LIN {X 98.327,Y 109.227,Z 74.500,A 180.000,B 0.000,C 180.000} C_DIS
LIN {X 98.684,Y 109.197,Z 74.500,A 180.000,B 0.000,C 180.000} C_DIS
LIN {X 98.863,Y 109.180,Z 74.500,A 180.000,B 0.000,C 180.000} C_DIS
LIN {X 99.042,Y 109.155,Z 74.500,A 180.000,B 0.000,C 180.000} C_DIS
LIN {X 99.221,Y 109.129,Z 74.500,A 180.000,B 0.000,C 180.000} C_DIS
LIN {X 99.399,Y 109.104,Z 74.500,A 180.000,B 0.000,C 180.000} C_DIS
LIN {X 99.578,Y 109.071,Z 74.500,A 180.000,B 0.000,C 180.000} C_DIS
LIN {X 99.672,Y 109.053,Z 74.500,A 180.000,B 0.000,C 180.000} C_DIS
LIN {X 99.936,Y 109.000,Z 74.500,A 180.000,B 0.000,C 180.000} C_DIS
LIN {X 100.114,Y 108.964,Z 74.500,A 180.000,B 0.000,C 180.000} C_DIS
LIN {X 100.293,Y 108.920,Z 74.500,A 180.000,B 0.000,C 180.000} C_DIS
LIN {X 100.651,Y 108.828,Z 74.500,A 180.000,B 0.000,C 180.000} C_DIS
LIN {X 100.829,Y 108.776,Z 74.500,A 180.000,B 0.000,C 180.000} C_DIS
LIN {X 101.187,Y 108.662,Z 74.500,A 180.000,B 0.000,C 180.000} C_DIS
LIN {X 101.366,Y 108.604,Z 74.500,A 180.000,B 0.000,C 180.000} C_DIS
LIN {X 101.545,Y 108.539,Z 74.500,A 180.000,B 0.000,C 180.000} C_DIS
LIN {X 101.902,Y 108.403,Z 74.500,A 180.000,B 0.000,C 180.000} C_DIS
LIN {X 102.060,Y 108.338,Z 74.500,A 180.000,B 0.000,C 180.000} C_DIS
LIN {X 102.459,Y 108.159,Z 74.500,A 180.000,B 0.000,C 180.000} C_DIS
LIN {X 102.617,Y 108.086,Z 74.500,A 180.000,B 0.000,C 180.000} C_DIS
LIN {X 102.796,Y 107.996,Z 74.500,A 180.000,B 0.000,C 180.000} C_DIS
LIN {X 102.975,Y 107.903,Z 74.500,A 180.000,B 0.000,C 180.000} C_DIS
LIN {X 103.153,Y 107.811,Z 74.500,A 180.000,B 0.000,C 180.000} C_DIS
LIN {X 103.171,Y 107.802,Z 74.500,A 180.000,B 0.000,C 180.000} C_DIS
LIN {X 103.332,Y 107.708,Z 74.500,A 180.000,B 0.000,C 180.000} C_DIS
LIN {X 103.511,Y 107.602,Z 74.500,A 180.000,B 0.000,C 180.000} C_DIS
LIN {X 103.690,Y 107.497,Z 74.500,A 180.000,B 0.000,C 180.000} C_DIS
LIN {X 103.773,Y 107.444,Z 74.500,A 180.000,B 0.000,C 180.000} C_DIS
LIN {X 103.869,Y 107.382,Z 74.500,A 180.000,B 0.000,C 180.000} C_DIS
LIN {X 104.226,Y 107.144,Z 74.500,A 180.000,B 0.000,C 180.000} C_DIS
LIN {X 104.310,Y 107.086,Z 74.500,A 180.000,B 0.000,C 180.000} C_DIS
LIN {X 104.405,Y 107.016,Z 74.500,A 180.000,B 0.000,C 180.000} C_DIS
LIN {X 104.584,Y 106.882,Z 74.500,A 180.000,B 0.000,C 180.000} C_DIS
LIN {X 104.762,Y 106.747,Z 74.500,A 180.000,B 0.000,C 180.000} C_DIS
LIN {X 104.786,Y 106.729,Z 74.500,A 180.000,B 0.000,C 180.000} C_DIS
LIN {X 104.941,Y 106.601,Z 74.500,A 180.000,B 0.000,C 180.000} C_DIS
LIN {X 105.299,Y 106.300,Z 74.500,A 180.000,B 0.000,C 180.000} C_DIS
LIN {X 105.417,Y 106.193,Z 74.500,A 180.000,B 0.000,C 180.000} C_DIS
LIN {X 105.656,Y 105.967,Z 74.500,A 180.000,B 0.000,C 180.000} C_DIS
LIN {X 105.794,Y 105.835,Z 74.500,A 180.000,B 0.000,C 180.000} C_DIS
LIN {X 105.835,Y 105.793,Z 74.500,A 180.000,B 0.000,C 180.000} C_DIS
LIN {X 105.965,Y 105.656,Z 74.500,A 180.000,B 0.000,C 180.000} C_DIS
LIN {X 106.134,Y 105.477,Z 74.500,A 180.000,B 0.000,C 180.000} C_DIS
LIN {X 106.193,Y 105.415,Z 74.500,A 180.000,B 0.000,C 180.000} C_DIS
LIN {X 106.300,Y 105.299,Z 74.500,A 180.000,B 0.000,C 180.000} C_DIS
LIN {X 106.371,Y 105.215,Z 74.500,A 180.000,B 0.000,C 180.000} C_DIS
LIN {X 106.603,Y 104.941,Z 74.500,A 180.000,B 0.000,C 180.000} C_DIS
LIN {X 106.729,Y 104.786,Z 74.500,A 180.000,B 0.000,C 180.000} C_DIS
LIN {X 107.015,Y 104.405,Z 74.500,A 180.000,B 0.000,C 180.000} C_DIS
LIN {X 107.086,Y 104.308,Z 74.500,A 180.000,B 0.000,C 180.000} C_DIS
LIN {X 107.144,Y 104.226,Z 74.500,A 180.000,B 0.000,C 180.000} C_DIS
LIN {X 107.265,Y 104.045,Z 74.500,A 180.000,B 0.000,C 180.000} C_DIS
LIN {X 107.383,Y 103.869,Z 74.500,A 180.000,B 0.000,C 180.000} C_DIS
LIN {X 107.444,Y 103.776,Z 74.500,A 180.000,B 0.000,C 180.000} C_DIS
LIN {X 107.497,Y 103.690,Z 74.500,A 180.000,B 0.000,C 180.000} C_DIS
LIN {X 107.708,Y 103.332,Z 74.500,A 180.000,B 0.000,C 180.000} C_DIS
LIN {X 107.802,Y 103.167,Z 74.500,A 180.000,B 0.000,C 180.000} C_DIS
LIN {X 107.809,Y 103.153,Z 74.500,A 180.000,B 0.000,C 180.000} C_DIS
LIN {X 107.903,Y 102.975,Z 74.500,A 180.000,B 0.000,C 180.000} C_DIS
LIN {X 107.995,Y 102.796,Z 74.500,A 180.000,B 0.000,C 180.000} C_DIS
LIN {X 108.087,Y 102.617,Z 74.500,A 180.000,B 0.000,C 180.000} C_DIS
LIN {X 108.159,Y 102.461,Z 74.500,A 180.000,B 0.000,C 180.000} C_DIS
LIN {X 108.249,Y 102.260,Z 74.500,A 180.000,B 0.000,C 180.000} C_DIS
LIN {X 108.329,Y 102.081,Z 74.500,A 180.000,B 0.000,C 180.000} C_DIS
LIN {X 108.338,Y 102.061,Z 74.500,A 180.000,B 0.000,C 180.000} C_DIS
LIN {X 108.402,Y 101.902,Z 74.500,A 180.000,B 0.000,C 180.000} C_DIS
LIN {X 108.470,Y 101.723,Z 74.500,A 180.000,B 0.000,C 180.000} C_DIS
LIN {X 108.538,Y 101.545,Z 74.500,A 180.000,B 0.000,C 180.000} C_DIS
LIN {X 108.605,Y 101.366,Z 74.500,A 180.000,B 0.000,C 180.000} C_DIS
LIN {X 108.663,Y 101.187,Z 74.500,A 180.000,B 0.000,C 180.000} C_DIS
LIN {X 108.720,Y 101.008,Z 74.500,A 180.000,B 0.000,C 180.000} C_DIS
LIN {X 108.777,Y 100.829,Z 74.500,A 180.000,B 0.000,C 180.000} C_DIS
LIN {X 108.826,Y 100.651,Z 74.500,A 180.000,B 0.000,C 180.000} C_DIS
LIN {X 108.919,Y 100.293,Z 74.500,A 180.000,B 0.000,C 180.000} C_DIS
LIN {X 108.964,Y 100.114,Z 74.500,A 180.000,B 0.000,C 180.000} C_DIS
LIN {X 109.002,Y 99.936,Z 74.500,A 180.000,B 0.000,C 180.000} C_DIS
LIN {X 109.073,Y 99.578,Z 74.500,A 180.000,B 0.000,C 180.000} C_DIS
LIN {X 109.103,Y 99.399,Z 74.500,A 180.000,B 0.000,C 180.000} C_DIS
LIN {X 109.154,Y 99.042,Z 74.500,A 180.000,B 0.000,C 180.000} C_DIS
LIN {X 109.178,Y 98.863,Z 74.500,A 180.000,B 0.000,C 180.000} C_DIS
LIN {X 109.197,Y 98.684,Z 74.500,A 180.000,B 0.000,C 180.000} C_DIS
LIN {X 109.232,Y 98.279,Z 74.500,A 180.000,B 0.000,C 180.000} C_DIS
LIN {X 109.241,Y 98.148,Z 74.500,A 180.000,B 0.000,C 180.000} C_DIS
LIN {X 109.247,Y 97.969,Z 74.500,A 180.000,B 0.000,C 180.000} C_DIS
LIN {X 109.252,Y 97.790,Z 74.500,A 180.000,B 0.000,C 180.000} C_DIS
LIN {X 109.257,Y 97.612,Z 74.500,A 180.000,B 0.000,C 180.000} C_DIS
LIN {X 109.257,Y 97.433,Z 74.500,A 180.000,B 0.000,C 180.000} C_DIS
LIN {X 109.253,Y 97.254,Z 74.500,A 180.000,B 0.000,C 180.000} C_DIS
LIN {X 109.248,Y 97.075,Z 74.500,A 180.000,B 0.000,C 180.000} C_DIS
LIN {X 109.243,Y 96.897,Z 74.500,A 180.000,B 0.000,C 180.000} C_DIS
LIN {X 109.232,Y 96.721,Z 74.500,A 180.000,B 0.000,C 180.000} C_DIS
LIN {X 109.201,Y 96.360,Z 74.500,A 180.000,B 0.000,C 180.000} C_DIS
LIN {X 109.184,Y 96.181,Z 74.500,A 180.000,B 0.000,C 180.000} C_DIS
LIN {X 109.160,Y 96.003,Z 74.500,A 180.000,B 0.000,C 180.000} C_DIS
LIN {X 109.110,Y 95.645,Z 74.500,A 180.000,B 0.000,C 180.000} C_DIS
LIN {X 109.081,Y 95.466,Z 74.500,A 180.000,B 0.000,C 180.000} C_DIS
LIN {X 109.053,Y 95.322,Z 74.500,A 180.000,B 0.000,C 180.000} C_DIS
LIN {X 109.010,Y 95.109,Z 74.500,A 180.000,B 0.000,C 180.000} C_DIS
LIN {X 108.974,Y 94.930,Z 74.500,A 180.000,B 0.000,C 180.000} C_DIS
LIN {X 108.930,Y 94.751,Z 74.500,A 180.000,B 0.000,C 180.000} C_DIS
LIN {X 108.838,Y 94.394,Z 74.500,A 180.000,B 0.000,C 180.000} C_DIS
LIN {X 108.791,Y 94.215,Z 74.500,A 180.000,B 0.000,C 180.000} C_DIS
LIN {X 108.734,Y 94.036,Z 74.500,A 180.000,B 0.000,C 180.000} C_DIS
LIN {X 108.677,Y 93.857,Z 74.500,A 180.000,B 0.000,C 180.000} C_DIS
LIN {X 108.620,Y 93.679,Z 74.500,A 180.000,B 0.000,C 180.000} C_DIS
LIN {X 108.555,Y 93.500,Z 74.500,A 180.000,B 0.000,C 180.000} C_DIS
LIN {X 108.419,Y 93.142,Z 74.500,A 180.000,B 0.000,C 180.000} C_DIS
LIN {X 108.348,Y 92.964,Z 74.500,A 180.000,B 0.000,C 180.000} C_DIS
LIN {X 108.338,Y 92.939,Z 74.500,A 180.000,B 0.000,C 180.000} C_DIS
LIN {X 108.269,Y 92.785,Z 74.500,A 180.000,B 0.000,C 180.000} C_DIS
LIN {X 108.159,Y 92.539,Z 74.500,A 180.000,B 0.000,C 180.000} C_DIS
LIN {X 108.109,Y 92.427,Z 74.500,A 180.000,B 0.000,C 180.000} C_DIS
LIN {X 108.018,Y 92.249,Z 74.500,A 180.000,B 0.000,C 180.000} C_DIS
LIN {X 107.926,Y 92.070,Z 74.500,A 180.000,B 0.000,C 180.000} C_DIS
LIN {X 107.833,Y 91.891,Z 74.500,A 180.000,B 0.000,C 180.000} C_DIS
LIN {X 107.802,Y 91.833,Z 74.500,A 180.000,B 0.000,C 180.000} C_DIS
LIN {X 107.734,Y 91.712,Z 74.500,A 180.000,B 0.000,C 180.000} C_DIS
LIN {X 107.523,Y 91.355,Z 74.500,A 180.000,B 0.000,C 180.000} C_DIS
LIN {X 107.444,Y 91.224,Z 74.500,A 180.000,B 0.000,C 180.000} C_DIS
LIN {X 107.413,Y 91.176,Z 74.500,A 180.000,B 0.000,C 180.000} C_DIS
LIN {X 107.174,Y 90.818,Z 74.500,A 180.000,B 0.000,C 180.000} C_DIS
LIN {X 107.086,Y 90.692,Z 74.500,A 180.000,B 0.000,C 180.000} C_DIS
LIN {X 107.048,Y 90.640,Z 74.500,A 180.000,B 0.000,C 180.000} C_DIS
LIN {X 106.914,Y 90.461,Z 74.500,A 180.000,B 0.000,C 180.000} C_DIS
LIN {X 106.729,Y 90.214,Z 74.500,A 180.000,B 0.000,C 180.000} C_DIS
LIN {X 106.640,Y 90.103,Z 74.500,A 180.000,B 0.000,C 180.000} C_DIS
LIN {X 106.338,Y 89.746,Z 74.500,A 180.000,B 0.000,C 180.000} C_DIS
LIN {X 106.193,Y 89.585,Z 74.500,A 180.000,B 0.000,C 180.000} C_DIS
LIN {X 106.176,Y 89.567,Z 74.500,A 180.000,B 0.000,C 180.000} C_DIS
LIN {X 106.007,Y 89.388,Z 74.500,A 180.000,B 0.000,C 180.000} C_DIS
LIN {X 105.838,Y 89.209,Z 74.500,A 180.000,B 0.000,C 180.000} C_DIS
LIN {X 105.835,Y 89.207,Z 74.500,A 180.000,B 0.000,C 180.000} C_DIS
LIN {X 105.656,Y 89.033,Z 74.500,A 180.000,B 0.000,C 180.000} C_DIS
LIN {X 105.464,Y 88.852,Z 74.500,A 180.000,B 0.000,C 180.000} C_DIS
LIN {X 105.299,Y 88.700,Z 74.500,A 180.000,B 0.000,C 180.000} C_DIS
LIN {X 104.941,Y 88.399,Z 74.500,A 180.000,B 0.000,C 180.000} C_DIS
LIN {X 104.841,Y 88.316,Z 74.500,A 180.000,B 0.000,C 180.000} C_DIS
LIN {X 104.762,Y 88.253,Z 74.500,A 180.000,B 0.000,C 180.000} C_DIS
LIN {X 104.608,Y 88.137,Z 74.500,A 180.000,B 0.000,C 180.000} C_DIS
LIN {X 104.371,Y 87.958,Z 74.500,A 180.000,B 0.000,C 180.000} C_DIS
LIN {X 104.226,Y 87.856,Z 74.500,A 180.000,B 0.000,C 180.000} C_DIS
LIN {X 103.869,Y 87.618,Z 74.500,A 180.000,B 0.000,C 180.000} C_DIS
LIN {X 103.843,Y 87.601,Z 74.500,A 180.000,B 0.000,C 180.000} C_DIS
LIN {X 103.690,Y 87.503,Z 74.500,A 180.000,B 0.000,C 180.000} C_DIS
LIN {X 103.552,Y 87.422,Z 74.500,A 180.000,B 0.000,C 180.000} C_DIS
LIN {X 103.249,Y 87.243,Z 74.500,A 180.000,B 0.000,C 180.000} C_DIS
LIN {X 103.153,Y 87.189,Z 74.500,A 180.000,B 0.000,C 180.000} C_DIS
LIN {X 102.975,Y 87.097,Z 74.500,A 180.000,B 0.000,C 180.000} C_DIS
LIN {X 102.796,Y 87.004,Z 74.500,A 180.000,B 0.000,C 180.000} C_DIS
LIN {X 102.617,Y 86.914,Z 74.500,A 180.000,B 0.000,C 180.000} C_DIS
LIN {X 102.556,Y 86.885,Z 74.500,A 180.000,B 0.000,C 180.000} C_DIS
LIN {X 102.438,Y 86.832,Z 74.500,A 180.000,B 0.000,C 180.000} C_DIS
LIN {X 102.191,Y 86.721,Z 74.500,A 180.000,B 0.000,C 180.000} C_DIS
; Link Move Starts
LIN {X 101.924,Y 86.603,Z 74.500,A 180.000,B 0.000,C 180.000} C_DIS
LIN {X 101.633,Y 86.492,Z 74.499,A 180.000,B 0.000,C 180.000} C_DIS
LIN {X 101.360,Y 86.390,Z 74.498,A 180.000,B 0.000,C 180.000} C_DIS
LIN {X 101.062,Y 86.294,Z 74.496,A 180.000,B 0.000,C 180.000} C_DIS
LIN {X 100.768,Y 86.200,Z 74.494,A 180.000,B 0.000,C 180.000} C_DIS
LIN {X 100.483,Y 86.123,Z 74.492,A 180.000,B 0.000,C 180.000} C_DIS
LIN {X 100.187,Y 86.045,Z 74.489,A 180.000,B 0.000,C 180.000} C_DIS
LIN {X 99.896,Y 85.983,Z 74.486,A 180.000,B 0.000,C 180.000} C_DIS
LIN {X 99.589,Y 85.920,Z 74.482,A 180.000,B 0.000,C 180.000} C_DIS
LIN {X 99.302,Y 85.870,Z 74.478,A 180.000,B 0.000,C 180.000} C_DIS
LIN {X 98.991,Y 85.824,Z 74.474,A 180.000,B 0.000,C 180.000} C_DIS
LIN {X 98.702,Y 85.788,Z 74.469,A 180.000,B 0.000,C 180.000} C_DIS
LIN {X 98.546,Y 85.773,Z 74.467,A 180.000,B 0.000,C 180.000} C_DIS
LIN {X 98.390,Y 85.759,Z 74.464,A 180.000,B 0.000,C 180.000} C_DIS
LIN {X 98.244,Y 85.746,Z 74.461,A 180.000,B 0.000,C 180.000} C_DIS
LIN {X 98.098,Y 85.736,Z 74.459,A 180.000,B 0.000,C 180.000} C_DIS
LIN {X 97.942,Y 85.729,Z 74.456,A 180.000,B 0.000,C 180.000} C_DIS
LIN {X 97.786,Y 85.724,Z 74.453,A 180.000,B 0.000,C 180.000} C_DIS
LIN {X 97.633,Y 85.718,Z 74.450,A 180.000,B 0.000,C 180.000} C_DIS
LIN {X 97.480,Y 85.714,Z 74.447,A 180.000,B 0.000,C 180.000} C_DIS
LIN {X 97.331,Y 85.716,Z 74.443,A 180.000,B 0.000,C 180.000} C_DIS
LIN {X 97.181,Y 85.719,Z 74.440,A 180.000,B 0.000,C 180.000} C_DIS
LIN {X 97.030,Y 85.721,Z 74.437,A 180.000,B 0.000,C 180.000} C_DIS
LIN {X 96.880,Y 85.725,Z 74.433,A 180.000,B 0.000,C 180.000} C_DIS
LIN {X 96.728,Y 85.733,Z 74.430,A 180.000,B 0.000,C 180.000} C_DIS
LIN {X 96.576,Y 85.744,Z 74.426,A 180.000,B 0.000,C 180.000} C_DIS
LIN {X 96.419,Y 85.756,Z 74.422,A 180.000,B 0.000,C 180.000} C_DIS
LIN {X 96.262,Y 85.767,Z 74.418,A 180.000,B 0.000,C 180.000} C_DIS
LIN {X 96.117,Y 85.781,Z 74.415,A 180.000,B 0.000,C 180.000} C_DIS
LIN {X 95.973,Y 85.799,Z 74.411,A 180.000,B 0.000,C 180.000} C_DIS
LIN {X 95.818,Y 85.819,Z 74.407,A 180.000,B 0.000,C 180.000} C_DIS
LIN {X 95.663,Y 85.839,Z 74.403,A 180.000,B 0.000,C 180.000} C_DIS
LIN {X 95.517,Y 85.860,Z 74.399,A 180.000,B 0.000,C 180.000} C_DIS
LIN {X 95.370,Y 85.886,Z 74.394,A 180.000,B 0.000,C 180.000} C_DIS
LIN {X 95.217,Y 85.915,Z 74.390,A 180.000,B 0.000,C 180.000} C_DIS
LIN {X 95.063,Y 85.943,Z 74.386,A 180.000,B 0.000,C 180.000} C_DIS
LIN {X 94.918,Y 85.970,Z 74.381,A 180.000,B 0.000,C 180.000} C_DIS
LIN {X 94.775,Y 86.001,Z 74.377,A 180.000,B 0.000,C 180.000} C_DIS
LIN {X 94.622,Y 86.038,Z 74.372,A 180.000,B 0.000,C 180.000} C_DIS
LIN {X 94.470,Y 86.075,Z 74.368,A 180.000,B 0.000,C 180.000} C_DIS
LIN {X 94.323,Y 86.110,Z 74.363,A 180.000,B 0.000,C 180.000} C_DIS
LIN {X 94.177,Y 86.150,Z 74.358,A 180.000,B 0.000,C 180.000} C_DIS
LIN {X 94.031,Y 86.194,Z 74.353,A 180.000,B 0.000,C 180.000} C_DIS
LIN {X 93.885,Y 86.238,Z 74.348,A 180.000,B 0.000,C 180.000} C_DIS
LIN {X 93.740,Y 86.282,Z 74.343,A 180.000,B 0.000,C 180.000} C_DIS
LIN {X 93.594,Y 86.327,Z 74.339,A 180.000,B 0.000,C 180.000} C_DIS
LIN {X 93.522,Y 86.351,Z 74.336,A 180.000,B 0.000,C 180.000} C_DIS
LIN {X 93.451,Y 86.377,Z 74.333,A 180.000,B 0.000,C 180.000} C_DIS
LIN {X 93.379,Y 86.403,Z 74.331,A 180.000,B 0.000,C 180.000} C_DIS
LIN {X 93.236,Y 86.455,Z 74.326,A 180.000,B 0.000,C 180.000} C_DIS
LIN {X 93.164,Y 86.481,Z 74.323,A 180.000,B 0.000,C 180.000} C_DIS
LIN {X 93.092,Y 86.508,Z 74.321,A 180.000,B 0.000,C 180.000} C_DIS
LIN {X 93.020,Y 86.534,Z 74.318,A 180.000,B 0.000,C 180.000} C_DIS
LIN {X 92.950,Y 86.561,Z 74.315,A 180.000,B 0.000,C 180.000} C_DIS
LIN {X 92.880,Y 86.591,Z 74.313,A 180.000,B 0.000,C 180.000} C_DIS
LIN {X 92.525,Y 86.743,Z 74.299,A 180.000,B 0.000,C 180.000} C_DIS
LIN {X 92.453,Y 86.774,Z 74.296,A 180.000,B 0.000,C 180.000} C_DIS
LIN {X 92.385,Y 86.804,Z 74.294,A 180.000,B 0.000,C 180.000} C_DIS
LIN {X 92.318,Y 86.835,Z 74.291,A 180.000,B 0.000,C 180.000} C_DIS
LIN {X 92.251,Y 86.867,Z 74.289,A 180.000,B 0.000,C 180.000} C_DIS
LIN {X 92.185,Y 86.899,Z 74.286,A 180.000,B 0.000,C 180.000} C_DIS
LIN {X 92.044,Y 86.969,Z 74.281,A 180.000,B 0.000,C 180.000} C_DIS
LIN {X 91.837,Y 87.072,Z 74.273,A 180.000,B 0.000,C 180.000} C_DIS
LIN {X 91.771,Y 87.106,Z 74.270,A 180.000,B 0.000,C 180.000} C_DIS
LIN {X 91.706,Y 87.141,Z 74.267,A 180.000,B 0.000,C 180.000} C_DIS
LIN {X 91.642,Y 87.177,Z 74.265,A 180.000,B 0.000,C 180.000} C_DIS
LIN {X 91.505,Y 87.255,Z 74.259,A 180.000,B 0.000,C 180.000} C_DIS
LIN {X 91.303,Y 87.370,Z 74.251,A 180.000,B 0.000,C 180.000} C_DIS
LIN {X 91.238,Y 87.407,Z 74.249,A 180.000,B 0.000,C 180.000} C_DIS
LIN {X 91.174,Y 87.446,Z 74.246,A 180.000,B 0.000,C 180.000} C_DIS
LIN {X 91.110,Y 87.485,Z 74.243,A 180.000,B 0.000,C 180.000} C_DIS
LIN {X 91.045,Y 87.527,Z 74.241,A 180.000,B 0.000,C 180.000} C_DIS
LIN {X 90.914,Y 87.611,Z 74.235,A 180.000,B 0.000,C 180.000} C_DIS
LIN {X 90.849,Y 87.654,Z 74.233,A 180.000,B 0.000,C 180.000} C_DIS
LIN {X 90.722,Y 87.735,Z 74.227,A 180.000,B 0.000,C 180.000} C_DIS
LIN {X 90.658,Y 87.776,Z 74.225,A 180.000,B 0.000,C 180.000} C_DIS
LIN {X 90.596,Y 87.819,Z 74.222,A 180.000,B 0.000,C 180.000} C_DIS
LIN {X 90.533,Y 87.864,Z 74.219,A 180.000,B 0.000,C 180.000} C_DIS
LIN {X 90.408,Y 87.955,Z 74.214,A 180.000,B 0.000,C 180.000} C_DIS
LIN {X 90.346,Y 88.000,Z 74.211,A 180.000,B 0.000,C 180.000} C_DIS
LIN {X 90.223,Y 88.090,Z 74.206,A 180.000,B 0.000,C 180.000} C_DIS
LIN {X 90.161,Y 88.134,Z 74.203,A 180.000,B 0.000,C 180.000} C_DIS
LIN {X 90.100,Y 88.180,Z 74.201,A 180.000,B 0.000,C 180.000} C_DIS
LIN {X 90.040,Y 88.228,Z 74.198,A 180.000,B 0.000,C 180.000} C_DIS
LIN {X 89.980,Y 88.276,Z 74.195,A 180.000,B 0.000,C 180.000} C_DIS
LIN {X 89.800,Y 88.423,Z 74.187,A 180.000,B 0.000,C 180.000} C_DIS
LIN {X 89.678,Y 88.523,Z 74.182,A 180.000,B 0.000,C 180.000} C_DIS
LIN {X 89.617,Y 88.573,Z 74.179,A 180.000,B 0.000,C 180.000} C_DIS
LIN {X 89.560,Y 88.620,Z 74.176,A 180.000,B 0.000,C 180.000} C_DIS
LIN {X 89.504,Y 88.669,Z 74.174,A 180.000,B 0.000,C 180.000} C_DIS
LIN {X 89.449,Y 88.719,Z 74.171,A 180.000,B 0.000,C 180.000} C_DIS
LIN {X 89.394,Y 88.770,Z 74.168,A 180.000,B 0.000,C 180.000} C_DIS
LIN {X 89.279,Y 88.875,Z 74.163,A 180.000,B 0.000,C 180.000} C_DIS
LIN {X 89.163,Y 88.981,Z 74.157,A 180.000,B 0.000,C 180.000} C_DIS
LIN {X 89.108,Y 89.032,Z 74.155,A 180.000,B 0.000,C 180.000} C_DIS
LIN {X 89.054,Y 89.084,Z 74.152,A 180.000,B 0.000,C 180.000} C_DIS
LIN {X 89.002,Y 89.138,Z 74.150,A 180.000,B 0.000,C 180.000} C_DIS
LIN {X 88.894,Y 89.248,Z 74.144,A 180.000,B 0.000,C 180.000} C_DIS
LIN {X 88.730,Y 89.417,Z 74.136,A 180.000,B 0.000,C 180.000} C_DIS
LIN {X 88.677,Y 89.470,Z 74.133,A 180.000,B 0.000,C 180.000} C_DIS
LIN {X 88.625,Y 89.524,Z 74.131,A 180.000,B 0.000,C 180.000} C_DIS
LIN {X 88.574,Y 89.578,Z 74.128,A 180.000,B 0.000,C 180.000} C_DIS
LIN {X 88.525,Y 89.634,Z 74.126,A 180.000,B 0.000,C 180.000} C_DIS
LIN {X 88.369,Y 89.812,Z 74.117,A 180.000,B 0.000,C 180.000} C_DIS
LIN {X 88.268,Y 89.927,Z 74.112,A 180.000,B 0.000,C 180.000} C_DIS
LIN {X 88.219,Y 89.984,Z 74.109,A 180.000,B 0.000,C 180.000} C_DIS
LIN {X 88.171,Y 90.041,Z 74.107,A 180.000,B 0.000,C 180.000} C_DIS
LIN {X 88.124,Y 90.099,Z 74.104,A 180.000,B 0.000,C 180.000} C_DIS
LIN {X 87.979,Y 90.286,Z 74.096,A 180.000,B 0.000,C 180.000} C_DIS
LIN {X 87.835,Y 90.470,Z 74.088,A 180.000,B 0.000,C 180.000} C_DIS
LIN {X 87.788,Y 90.532,Z 74.085,A 180.000,B 0.000,C 180.000} C_DIS
LIN {X 87.741,Y 90.594,Z 74.082,A 180.000,B 0.000,C 180.000} C_DIS
LIN {X 87.697,Y 90.656,Z 74.080,A 180.000,B 0.000,C 180.000} C_DIS
LIN {X 87.653,Y 90.718,Z 74.077,A 180.000,B 0.000,C 180.000} C_DIS
LIN {X 87.433,Y 91.037,Z 74.063,A 180.000,B 0.000,C 180.000} C_DIS
LIN {X 87.389,Y 91.101,Z 74.061,A 180.000,B 0.000,C 180.000} C_DIS
LIN {X 87.347,Y 91.164,Z 74.058,A 180.000,B 0.000,C 180.000} C_DIS
LIN {X 87.308,Y 91.229,Z 74.055,A 180.000,B 0.000,C 180.000} C_DIS
LIN {X 87.106,Y 91.558,Z 74.042,A 180.000,B 0.000,C 180.000} C_DIS
LIN {X 87.065,Y 91.625,Z 74.039,A 180.000,B 0.000,C 180.000} C_DIS
LIN {X 87.027,Y 91.691,Z 74.037,A 180.000,B 0.000,C 180.000} C_DIS
LIN {X 86.990,Y 91.756,Z 74.034,A 180.000,B 0.000,C 180.000} C_DIS
LIN {X 86.953,Y 91.822,Z 74.031,A 180.000,B 0.000,C 180.000} C_DIS
LIN {X 86.733,Y 92.233,Z 74.015,A 180.000,B 0.000,C 180.000} C_DIS
LIN {X 86.698,Y 92.300,Z 74.012,A 180.000,B 0.000,C 180.000} C_DIS
LIN {X 86.665,Y 92.368,Z 74.010,A 180.000,B 0.000,C 180.000} C_DIS
LIN {X 86.468,Y 92.789,Z 73.993,A 180.000,B 0.000,C 180.000} C_DIS
LIN {X 86.436,Y 92.858,Z 73.991,A 180.000,B 0.000,C 180.000} C_DIS
LIN {X 86.406,Y 92.928,Z 73.988,A 180.000,B 0.000,C 180.000} C_DIS
LIN {X 86.377,Y 92.999,Z 73.986,A 180.000,B 0.000,C 180.000} C_DIS
LIN {X 86.348,Y 93.071,Z 73.983,A 180.000,B 0.000,C 180.000} C_DIS
LIN {X 86.204,Y 93.432,Z 73.969,A 180.000,B 0.000,C 180.000} C_DIS
LIN {X 86.175,Y 93.502,Z 73.967,A 180.000,B 0.000,C 180.000} C_DIS
LIN {X 86.149,Y 93.574,Z 73.964,A 180.000,B 0.000,C 180.000} C_DIS
LIN {X 86.123,Y 93.648,Z 73.961,A 180.000,B 0.000,C 180.000} C_DIS
LIN {X 85.975,Y 94.089,Z 73.945,A 180.000,B 0.000,C 180.000} C_DIS
LIN {X 85.952,Y 94.162,Z 73.942,A 180.000,B 0.000,C 180.000} C_DIS
LIN {X 85.930,Y 94.237,Z 73.940,A 180.000,B 0.000,C 180.000} C_DIS
LIN {X 85.806,Y 94.690,Z 73.923,A 180.000,B 0.000,C 180.000} C_DIS
LIN {X 85.785,Y 94.766,Z 73.920,A 180.000,B 0.000,C 180.000} C_DIS
LIN {X 85.765,Y 94.839,Z 73.918,A 180.000,B 0.000,C 180.000} C_DIS
LIN {X 85.748,Y 94.913,Z 73.915,A 180.000,B 0.000,C 180.000} C_DIS
LIN {X 85.650,Y 95.370,Z 73.899,A 180.000,B 0.000,C 180.000} C_DIS
LIN {X 85.634,Y 95.444,Z 73.896,A 180.000,B 0.000,C 180.000} C_DIS
LIN {X 85.620,Y 95.519,Z 73.893,A 180.000,B 0.000,C 180.000} C_DIS
LIN {X 85.608,Y 95.595,Z 73.891,A 180.000,B 0.000,C 180.000} C_DIS
LIN {X 85.584,Y 95.748,Z 73.885,A 180.000,B 0.000,C 180.000} C_DIS
LIN {X 85.547,Y 95.981,Z 73.877,A 180.000,B 0.000,C 180.000} C_DIS
LIN {X 85.536,Y 96.057,Z 73.874,A 180.000,B 0.000,C 180.000} C_DIS
LIN {X 85.525,Y 96.132,Z 73.872,A 180.000,B 0.000,C 180.000} C_DIS
LIN {X 85.515,Y 96.208,Z 73.869,A 180.000,B 0.000,C 180.000} C_DIS
LIN {X 85.507,Y 96.284,Z 73.866,A 180.000,B 0.000,C 180.000} C_DIS
LIN {X 85.483,Y 96.519,Z 73.858,A 180.000,B 0.000,C 180.000} C_DIS
LIN {X 85.467,Y 96.674,Z 73.853,A 180.000,B 0.000,C 180.000} C_DIS
LIN {X 85.460,Y 96.750,Z 73.850,A 180.000,B 0.000,C 180.000} C_DIS
LIN {X 85.453,Y 96.827,Z 73.847,A 180.000,B 0.000,C 180.000} C_DIS
LIN {X 85.449,Y 96.904,Z 73.845,A 180.000,B 0.000,C 180.000} C_DIS
LIN {X 85.442,Y 97.060,Z 73.839,A 180.000,B 0.000,C 180.000} C_DIS
LIN {X 85.428,Y 97.371,Z 73.828,A 180.000,B 0.000,C 180.000} C_DIS
LIN {X 85.426,Y 97.449,Z 73.826,A 180.000,B 0.000,C 180.000} C_DIS
LIN {X 85.424,Y 97.526,Z 73.823,A 180.000,B 0.000,C 180.000} C_DIS
LIN {X 85.424,Y 97.604,Z 73.820,A 180.000,B 0.000,C 180.000} C_DIS
LIN {X 85.425,Y 97.682,Z 73.818,A 180.000,B 0.000,C 180.000} C_DIS
LIN {X 85.429,Y 98.070,Z 73.804,A 180.000,B 0.000,C 180.000} C_DIS
LIN {X 85.430,Y 98.147,Z 73.801,A 180.000,B 0.000,C 180.000} C_DIS
LIN {X 85.434,Y 98.225,Z 73.799,A 180.000,B 0.000,C 180.000} C_DIS
LIN {X 85.439,Y 98.304,Z 73.796,A 180.000,B 0.000,C 180.000} C_DIS
LIN {X 85.455,Y 98.538,Z 73.788,A 180.000,B 0.000,C 180.000} C_DIS
LIN {X 85.465,Y 98.694,Z 73.782,A 180.000,B 0.000,C 180.000} C_DIS
LIN {X 85.471,Y 98.773,Z 73.779,A 180.000,B 0.000,C 180.000} C_DIS
LIN {X 85.478,Y 98.849,Z 73.777,A 180.000,B 0.000,C 180.000} C_DIS
LIN {X 85.486,Y 98.926,Z 73.774,A 180.000,B 0.000,C 180.000} C_DIS
LIN {X 85.495,Y 99.003,Z 73.771,A 180.000,B 0.000,C 180.000} C_DIS
LIN {X 85.505,Y 99.080,Z 73.769,A 180.000,B 0.000,C 180.000} C_DIS
LIN {X 85.524,Y 99.236,Z 73.763,A 180.000,B 0.000,C 180.000} C_DIS
LIN {X 85.553,Y 99.468,Z 73.755,A 180.000,B 0.000,C 180.000} C_DIS
LIN {X 85.564,Y 99.545,Z 73.752,A 180.000,B 0.000,C 180.000} C_DIS
LIN {X 85.577,Y 99.621,Z 73.750,A 180.000,B 0.000,C 180.000} C_DIS
LIN {X 85.591,Y 99.697,Z 73.747,A 180.000,B 0.000,C 180.000} C_DIS
LIN {X 85.619,Y 99.852,Z 73.741,A 180.000,B 0.000,C 180.000} C_DIS
LIN {X 85.661,Y 100.083,Z 73.733,A 180.000,B 0.000,C 180.000} C_DIS
LIN {X 85.675,Y 100.159,Z 73.730,A 180.000,B 0.000,C 180.000} C_DIS
LIN {X 85.692,Y 100.235,Z 73.728,A 180.000,B 0.000,C 180.000} C_DIS
LIN {X 85.710,Y 100.310,Z 73.725,A 180.000,B 0.000,C 180.000} C_DIS
LIN {X 85.729,Y 100.386,Z 73.722,A 180.000,B 0.000,C 180.000} C_DIS
LIN {X 85.765,Y 100.539,Z 73.717,A 180.000,B 0.000,C 180.000} C_DIS
LIN {X 85.784,Y 100.616,Z 73.714,A 180.000,B 0.000,C 180.000} C_DIS
LIN {X 85.820,Y 100.768,Z 73.709,A 180.000,B 0.000,C 180.000} C_DIS
LIN {X 85.839,Y 100.843,Z 73.706,A 180.000,B 0.000,C 180.000} C_DIS
LIN {X 85.859,Y 100.919,Z 73.703,A 180.000,B 0.000,C 180.000} C_DIS
LIN {X 85.881,Y 100.994,Z 73.700,A 180.000,B 0.000,C 180.000} C_DIS
LIN {X 85.927,Y 101.143,Z 73.695,A 180.000,B 0.000,C 180.000} C_DIS
LIN {X 85.994,Y 101.368,Z 73.687,A 180.000,B 0.000,C 180.000} C_DIS
LIN {X 86.017,Y 101.443,Z 73.684,A 180.000,B 0.000,C 180.000} C_DIS
LIN {X 86.041,Y 101.517,Z 73.681,A 180.000,B 0.000,C 180.000} C_DIS
LIN {X 86.067,Y 101.591,Z 73.679,A 180.000,B 0.000,C 180.000} C_DIS
LIN {X 86.094,Y 101.664,Z 73.676,A 180.000,B 0.000,C 180.000} C_DIS
LIN {X 86.121,Y 101.738,Z 73.674,A 180.000,B 0.000,C 180.000} C_DIS
LIN {X 86.147,Y 101.811,Z 73.671,A 180.000,B 0.000,C 180.000} C_DIS
LIN {X 86.174,Y 101.885,Z 73.668,A 180.000,B 0.000,C 180.000} C_DIS
LIN {X 86.201,Y 101.958,Z 73.666,A 180.000,B 0.000,C 180.000} C_DIS
LIN {X 86.228,Y 102.032,Z 73.663,A 180.000,B 0.000,C 180.000} C_DIS
LIN {X 86.255,Y 102.105,Z 73.661,A 180.000,B 0.000,C 180.000} C_DIS
LIN {X 86.283,Y 102.178,Z 73.658,A 180.000,B 0.000,C 180.000} C_DIS
LIN {X 86.313,Y 102.250,Z 73.655,A 180.000,B 0.000,C 180.000} C_DIS
LIN {X 86.344,Y 102.322,Z 73.653,A 180.000,B 0.000,C 180.000} C_DIS
LIN {X 86.375,Y 102.394,Z 73.650,A 180.000,B 0.000,C 180.000} C_DIS
LIN {X 86.437,Y 102.539,Z 73.645,A 180.000,B 0.000,C 180.000} C_DIS
LIN {X 86.499,Y 102.683,Z 73.641,A 180.000,B 0.000,C 180.000} C_DIS
LIN {X 86.564,Y 102.825,Z 73.636,A 180.000,B 0.000,C 180.000} C_DIS
LIN {X 86.633,Y 102.965,Z 73.631,A 180.000,B 0.000,C 180.000} C_DIS
LIN {X 86.704,Y 103.105,Z 73.626,A 180.000,B 0.000,C 180.000} C_DIS
LIN {X 86.774,Y 103.246,Z 73.622,A 180.000,B 0.000,C 180.000} C_DIS
LIN {X 86.845,Y 103.385,Z 73.617,A 180.000,B 0.000,C 180.000} C_DIS
LIN {X 86.921,Y 103.522,Z 73.613,A 180.000,B 0.000,C 180.000} C_DIS
LIN {X 86.999,Y 103.658,Z 73.608,A 180.000,B 0.000,C 180.000} C_DIS
LIN {X 87.077,Y 103.795,Z 73.604,A 180.000,B 0.000,C 180.000} C_DIS
LIN {X 87.155,Y 103.931,Z 73.599,A 180.000,B 0.000,C 180.000} C_DIS
LIN {X 87.237,Y 104.063,Z 73.595,A 180.000,B 0.000,C 180.000} C_DIS
LIN {X 87.323,Y 104.195,Z 73.591,A 180.000,B 0.000,C 180.000} C_DIS
LIN {X 87.409,Y 104.327,Z 73.587,A 180.000,B 0.000,C 180.000} C_DIS
LIN {X 87.495,Y 104.459,Z 73.583,A 180.000,B 0.000,C 180.000} C_DIS
LIN {X 87.583,Y 104.588,Z 73.579,A 180.000,B 0.000,C 180.000} C_DIS
LIN {X 87.676,Y 104.715,Z 73.575,A 180.000,B 0.000,C 180.000} C_DIS
LIN {X 87.769,Y 104.842,Z 73.572,A 180.000,B 0.000,C 180.000} C_DIS
LIN {X 87.862,Y 104.969,Z 73.568,A 180.000,B 0.000,C 180.000} C_DIS
LIN {X 87.956,Y 105.095,Z 73.564,A 180.000,B 0.000,C 180.000} C_DIS
LIN {X 88.054,Y 105.217,Z 73.561,A 180.000,B 0.000,C 180.000} C_DIS
LIN {X 88.154,Y 105.338,Z 73.557,A 180.000,B 0.000,C 180.000} C_DIS
LIN {X 88.254,Y 105.459,Z 73.554,A 180.000,B 0.000,C 180.000} C_DIS
LIN {X 88.355,Y 105.580,Z 73.551,A 180.000,B 0.000,C 180.000} C_DIS
LIN {X 88.460,Y 105.697,Z 73.548,A 180.000,B 0.000,C 180.000} C_DIS
LIN {X 88.566,Y 105.812,Z 73.545,A 180.000,B 0.000,C 180.000} C_DIS
LIN {X 88.674,Y 105.928,Z 73.542,A 180.000,B 0.000,C 180.000} C_DIS
LIN {X 88.781,Y 106.043,Z 73.539,A 180.000,B 0.000,C 180.000} C_DIS
LIN {X 88.889,Y 106.157,Z 73.536,A 180.000,B 0.000,C 180.000} C_DIS
LIN {X 89.002,Y 106.266,Z 73.533,A 180.000,B 0.000,C 180.000} C_DIS
LIN {X 89.115,Y 106.376,Z 73.531,A 180.000,B 0.000,C 180.000} C_DIS
LIN {X 89.229,Y 106.485,Z 73.528,A 180.000,B 0.000,C 180.000} C_DIS
LIN {X 89.461,Y 106.696,Z 73.523,A 180.000,B 0.000,C 180.000} C_DIS
LIN {X 89.701,Y 106.901,Z 73.519,A 180.000,B 0.000,C 180.000} C_DIS
LIN {X 89.942,Y 107.102,Z 73.515,A 180.000,B 0.000,C 180.000} C_DIS
LIN {X 90.193,Y 107.293,Z 73.512,A 180.000,B 0.000,C 180.000} C_DIS
LIN {X 90.445,Y 107.482,Z 73.509,A 180.000,B 0.000,C 180.000} C_DIS
LIN {X 90.706,Y 107.658,Z 73.506,A 180.000,B 0.000,C 180.000} C_DIS
LIN {X 90.968,Y 107.833,Z 73.504,A 180.000,B 0.000,C 180.000} C_DIS
LIN {X 91.237,Y 107.996,Z 73.502,A 180.000,B 0.000,C 180.000} C_DIS
LIN {X 91.508,Y 108.157,Z 73.501,A 180.000,B 0.000,C 180.000} C_DIS
LIN {X 91.785,Y 108.306,Z 73.500,A 180.000,B 0.000,C 180.000} C_DIS
LIN {X 92.065,Y 108.451,Z 73.500,A 180.000,B 0.000,C 180.000} C_DIS
LIN {X 92.082,Y 108.460,Z 73.500,A 180.000,B 0.000,C 180.000} C_DIS
; Cutting Move Starts
LIN {X 92.197,Y 108.517,Z 73.500,A 180.000,B 0.000,C 180.000} C_DIS
LIN {X 92.249,Y 108.541,Z 73.500,A 180.000,B 0.000,C 180.000} C_DIS
LIN {X 92.427,Y 108.622,Z 73.500,A 180.000,B 0.000,C 180.000} C_DIS
LIN {X 92.606,Y 108.702,Z 73.500,A 180.000,B 0.000,C 180.000} C_DIS
LIN {X 92.785,Y 108.782,Z 73.500,A 180.000,B 0.000,C 180.000} C_DIS
LIN {X 92.964,Y 108.853,Z 73.500,A 180.000,B 0.000,C 180.000} C_DIS
LIN {X 93.321,Y 108.989,Z 73.500,A 180.000,B 0.000,C 180.000} C_DIS
LIN {X 93.498,Y 109.053,Z 73.500,A 180.000,B 0.000,C 180.000} C_DIS
LIN {X 93.500,Y 109.053,Z 73.500,A 180.000,B 0.000,C 180.000} C_DIS
LIN {X 93.679,Y 109.111,Z 73.500,A 180.000,B 0.000,C 180.000} C_DIS
LIN {X 94.057,Y 109.232,Z 73.500,A 180.000,B 0.000,C 180.000} C_DIS
LIN {X 94.215,Y 109.277,Z 73.500,A 180.000,B 0.000,C 180.000} C_DIS
LIN {X 94.573,Y 109.369,Z 73.500,A 180.000,B 0.000,C 180.000} C_DIS
LIN {X 94.734,Y 109.410,Z 73.500,A 180.000,B 0.000,C 180.000} C_DIS
LIN {X 94.751,Y 109.415,Z 73.500,A 180.000,B 0.000,C 180.000} C_DIS
LIN {X 94.930,Y 109.451,Z 73.500,A 180.000,B 0.000,C 180.000} C_DIS
LIN {X 95.288,Y 109.523,Z 73.500,A 180.000,B 0.000,C 180.000} C_DIS
LIN {X 95.466,Y 109.557,Z 73.500,A 180.000,B 0.000,C 180.000} C_DIS
LIN {X 95.645,Y 109.583,Z 73.500,A 180.000,B 0.000,C 180.000} C_DIS
LIN {X 96.003,Y 109.634,Z 73.500,A 180.000,B 0.000,C 180.000} C_DIS
LIN {X 96.181,Y 109.656,Z 73.500,A 180.000,B 0.000,C 180.000} C_DIS
LIN {X 96.360,Y 109.671,Z 73.500,A 180.000,B 0.000,C 180.000} C_DIS
LIN {X 96.539,Y 109.686,Z 73.500,A 180.000,B 0.000,C 180.000} C_DIS
LIN {X 96.718,Y 109.701,Z 73.500,A 180.000,B 0.000,C 180.000} C_DIS
LIN {X 96.897,Y 109.712,Z 73.500,A 180.000,B 0.000,C 180.000} C_DIS
LIN {X 97.075,Y 109.717,Z 73.500,A 180.000,B 0.000,C 180.000} C_DIS
LIN {X 97.433,Y 109.727,Z 73.500,A 180.000,B 0.000,C 180.000} C_DIS
LIN {X 97.612,Y 109.726,Z 73.500,A 180.000,B 0.000,C 180.000} C_DIS
LIN {X 97.969,Y 109.716,Z 73.500,A 180.000,B 0.000,C 180.000} C_DIS
LIN {X 98.148,Y 109.710,Z 73.500,A 180.000,B 0.000,C 180.000} C_DIS
LIN {X 98.327,Y 109.697,Z 73.500,A 180.000,B 0.000,C 180.000} C_DIS
LIN {X 98.684,Y 109.667,Z 73.500,A 180.000,B 0.000,C 180.000} C_DIS
LIN {X 98.863,Y 109.651,Z 73.500,A 180.000,B 0.000,C 180.000} C_DIS
LIN {X 99.042,Y 109.628,Z 73.500,A 180.000,B 0.000,C 180.000} C_DIS
LIN {X 99.399,Y 109.577,Z 73.500,A 180.000,B 0.000,C 180.000} C_DIS
LIN {X 99.578,Y 109.549,Z 73.500,A 180.000,B 0.000,C 180.000} C_DIS
LIN {X 99.757,Y 109.514,Z 73.500,A 180.000,B 0.000,C 180.000} C_DIS
LIN {X 100.114,Y 109.443,Z 73.500,A 180.000,B 0.000,C 180.000} C_DIS
LIN {X 100.266,Y 109.410,Z 73.500,A 180.000,B 0.000,C 180.000} C_DIS
LIN {X 100.293,Y 109.404,Z 73.500,A 180.000,B 0.000,C 180.000} C_DIS
LIN {X 100.472,Y 109.358,Z 73.500,A 180.000,B 0.000,C 180.000} C_DIS
LIN {X 100.651,Y 109.312,Z 73.500,A 180.000,B 0.000,C 180.000} C_DIS
LIN {X 100.829,Y 109.265,Z 73.500,A 180.000,B 0.000,C 180.000} C_DIS
LIN {X 100.943,Y 109.232,Z 73.500,A 180.000,B 0.000,C 180.000} C_DIS
LIN {X 101.366,Y 109.097,Z 73.500,A 180.000,B 0.000,C 180.000} C_DIS
LIN {X 101.502,Y 109.053,Z 73.500,A 180.000,B 0.000,C 180.000} C_DIS
LIN {X 101.545,Y 109.039,Z 73.500,A 180.000,B 0.000,C 180.000} C_DIS
LIN {X 101.723,Y 108.972,Z 73.500,A 180.000,B 0.000,C 180.000} C_DIS
LIN {X 102.081,Y 108.836,Z 73.500,A 180.000,B 0.000,C 180.000} C_DIS
LIN {X 102.260,Y 108.762,Z 73.500,A 180.000,B 0.000,C 180.000} C_DIS
LIN {X 102.617,Y 108.602,Z 73.500,A 180.000,B 0.000,C 180.000} C_DIS
LIN {X 102.796,Y 108.520,Z 73.500,A 180.000,B 0.000,C 180.000} C_DIS
LIN {X 102.803,Y 108.517,Z 73.500,A 180.000,B 0.000,C 180.000} C_DIS
LIN {X 102.975,Y 108.431,Z 73.500,A 180.000,B 0.000,C 180.000} C_DIS
LIN {X 103.332,Y 108.246,Z 73.500,A 180.000,B 0.000,C 180.000} C_DIS
LIN {X 103.490,Y 108.159,Z 73.500,A 180.000,B 0.000,C 180.000} C_DIS
LIN {X 103.869,Y 107.935,Z 73.500,A 180.000,B 0.000,C 180.000} C_DIS
LIN {X 104.047,Y 107.825,Z 73.500,A 180.000,B 0.000,C 180.000} C_DIS
LIN {X 104.085,Y 107.802,Z 73.500,A 180.000,B 0.000,C 180.000} C_DIS
LIN {X 104.226,Y 107.707,Z 73.500,A 180.000,B 0.000,C 180.000} C_DIS
LIN {X 104.405,Y 107.588,Z 73.500,A 180.000,B 0.000,C 180.000} C_DIS
LIN {X 104.584,Y 107.467,Z 73.500,A 180.000,B 0.000,C 180.000} C_DIS
LIN {X 104.615,Y 107.444,Z 73.500,A 180.000,B 0.000,C 180.000} C_DIS
LIN {X 104.762,Y 107.334,Z 73.500,A 180.000,B 0.000,C 180.000} C_DIS
LIN {X 104.941,Y 107.199,Z 73.500,A 180.000,B 0.000,C 180.000} C_DIS
LIN {X 105.090,Y 107.086,Z 73.500,A 180.000,B 0.000,C 180.000} C_DIS
LIN {X 105.120,Y 107.062,Z 73.500,A 180.000,B 0.000,C 180.000} C_DIS
LIN {X 105.299,Y 106.913,Z 73.500,A 180.000,B 0.000,C 180.000} C_DIS
LIN {X 105.517,Y 106.729,Z 73.500,A 180.000,B 0.000,C 180.000} C_DIS
LIN {X 105.656,Y 106.610,Z 73.500,A 180.000,B 0.000,C 180.000} C_DIS
LIN {X 105.721,Y 106.550,Z 73.500,A 180.000,B 0.000,C 180.000} C_DIS
LIN {X 106.014,Y 106.273,Z 73.500,A 180.000,B 0.000,C 180.000} C_DIS
LIN {X 106.099,Y 106.193,Z 73.500,A 180.000,B 0.000,C 180.000} C_DIS
LIN {X 106.193,Y 106.097,Z 73.500,A 180.000,B 0.000,C 180.000} C_DIS
LIN {X 106.441,Y 105.835,Z 73.500,A 180.000,B 0.000,C 180.000} C_DIS
LIN {X 106.550,Y 105.719,Z 73.500,A 180.000,B 0.000,C 180.000} C_DIS
LIN {X 106.609,Y 105.656,Z 73.500,A 180.000,B 0.000,C 180.000} C_DIS
LIN {X 106.729,Y 105.518,Z 73.500,A 180.000,B 0.000,C 180.000} C_DIS
LIN {X 106.914,Y 105.299,Z 73.500,A 180.000,B 0.000,C 180.000} C_DIS
LIN {X 107.063,Y 105.120,Z 73.500,A 180.000,B 0.000,C 180.000} C_DIS
LIN {X 107.086,Y 105.090,Z 73.500,A 180.000,B 0.000,C 180.000} C_DIS
LIN {X 107.198,Y 104.941,Z 73.500,A 180.000,B 0.000,C 180.000} C_DIS
LIN {X 107.333,Y 104.762,Z 73.500,A 180.000,B 0.000,C 180.000} C_DIS
LIN {X 107.444,Y 104.613,Z 73.500,A 180.000,B 0.000,C 180.000} C_DIS
LIN {X 107.465,Y 104.584,Z 73.500,A 180.000,B 0.000,C 180.000} C_DIS
LIN {X 107.588,Y 104.405,Z 73.500,A 180.000,B 0.000,C 180.000} C_DIS
LIN {X 107.802,Y 104.085,Z 73.500,A 180.000,B 0.000,C 180.000} C_DIS
LIN {X 107.827,Y 104.047,Z 73.500,A 180.000,B 0.000,C 180.000} C_DIS
LIN {X 107.935,Y 103.869,Z 73.500,A 180.000,B 0.000,C 180.000} C_DIS
LIN {X 108.146,Y 103.511,Z 73.500,A 180.000,B 0.000,C 180.000} C_DIS
LIN {X 108.159,Y 103.489,Z 73.500,A 180.000,B 0.000,C 180.000} C_DIS
LIN {X 108.245,Y 103.332,Z 73.500,A 180.000,B 0.000,C 180.000} C_DIS
LIN {X 108.338,Y 103.153,Z 73.500,A 180.000,B 0.000,C 180.000} C_DIS
LIN {X 108.430,Y 102.975,Z 73.500,A 180.000,B 0.000,C 180.000} C_DIS
LIN {X 108.517,Y 102.806,Z 73.500,A 180.000,B 0.000,C 180.000} C_DIS
LIN {X 108.521,Y 102.796,Z 73.500,A 180.000,B 0.000,C 180.000} C_DIS
LIN {X 108.602,Y 102.617,Z 73.500,A 180.000,B 0.000,C 180.000} C_DIS
LIN {X 108.695,Y 102.409,Z 73.500,A 180.000,B 0.000,C 180.000} C_DIS
LIN {X 108.762,Y 102.260,Z 73.500,A 180.000,B 0.000,C 180.000} C_DIS
LIN {X 108.835,Y 102.081,Z 73.500,A 180.000,B 0.000,C 180.000} C_DIS
LIN {X 108.874,Y 101.978,Z 73.500,A 180.000,B 0.000,C 180.000} C_DIS
LIN {X 108.971,Y 101.723,Z 73.500,A 180.000,B 0.000,C 180.000} C_DIS
LIN {X 109.039,Y 101.545,Z 73.500,A 180.000,B 0.000,C 180.000} C_DIS
LIN {X 109.053,Y 101.505,Z 73.500,A 180.000,B 0.000,C 180.000} C_DIS
LIN {X 109.098,Y 101.366,Z 73.500,A 180.000,B 0.000,C 180.000} C_DIS
LIN {X 109.212,Y 101.008,Z 73.500,A 180.000,B 0.000,C 180.000} C_DIS
LIN {X 109.232,Y 100.946,Z 73.500,A 180.000,B 0.000,C 180.000} C_DIS
LIN {X 109.264,Y 100.829,Z 73.500,A 180.000,B 0.000,C 180.000} C_DIS
LIN {X 109.356,Y 100.472,Z 73.500,A 180.000,B 0.000,C 180.000} C_DIS
LIN {X 109.402,Y 100.293,Z 73.500,A 180.000,B 0.000,C 180.000} C_DIS
LIN {X 109.410,Y 100.262,Z 73.500,A 180.000,B 0.000,C 180.000} C_DIS
LIN {X 109.444,Y 100.114,Z 73.500,A 180.000,B 0.000,C 180.000} C_DIS
LIN {X 109.515,Y 99.757,Z 73.500,A 180.000,B 0.000,C 180.000} C_DIS
LIN {X 109.550,Y 99.578,Z 73.500,A 180.000,B 0.000,C 180.000} C_DIS
LIN {X 109.576,Y 99.399,Z 73.500,A 180.000,B 0.000,C 180.000} C_DIS
LIN {X 109.627,Y 99.042,Z 73.500,A 180.000,B 0.000,C 180.000} C_DIS
LIN {X 109.651,Y 98.863,Z 73.500,A 180.000,B 0.000,C 180.000} C_DIS
LIN {X 109.668,Y 98.684,Z 73.500,A 180.000,B 0.000,C 180.000} C_DIS
LIN {X 109.698,Y 98.327,Z 73.500,A 180.000,B 0.000,C 180.000} C_DIS
LIN {X 109.710,Y 98.148,Z 73.500,A 180.000,B 0.000,C 180.000} C_DIS
LIN {X 109.715,Y 97.969,Z 73.500,A 180.000,B 0.000,C 180.000} C_DIS
LIN {X 109.725,Y 97.612,Z 73.500,A 180.000,B 0.000,C 180.000} C_DIS
LIN {X 109.726,Y 97.433,Z 73.500,A 180.000,B 0.000,C 180.000} C_DIS
LIN {X 109.722,Y 97.254,Z 73.500,A 180.000,B 0.000,C 180.000} C_DIS
LIN {X 109.712,Y 96.897,Z 73.500,A 180.000,B 0.000,C 180.000} C_DIS
LIN {X 109.701,Y 96.718,Z 73.500,A 180.000,B 0.000,C 180.000} C_DIS
LIN {X 109.671,Y 96.360,Z 73.500,A 180.000,B 0.000,C 180.000} C_DIS
LIN {X 109.656,Y 96.181,Z 73.500,A 180.000,B 0.000,C 180.000} C_DIS
LIN {X 109.633,Y 96.003,Z 73.500,A 180.000,B 0.000,C 180.000} C_DIS
LIN {X 109.583,Y 95.645,Z 73.500,A 180.000,B 0.000,C 180.000} C_DIS
LIN {X 109.557,Y 95.466,Z 73.500,A 180.000,B 0.000,C 180.000} C_DIS
LIN {X 109.524,Y 95.288,Z 73.500,A 180.000,B 0.000,C 180.000} C_DIS
LIN {X 109.452,Y 94.930,Z 73.500,A 180.000,B 0.000,C 180.000} C_DIS
LIN {X 109.414,Y 94.751,Z 73.500,A 180.000,B 0.000,C 180.000} C_DIS
LIN {X 109.410,Y 94.738,Z 73.500,A 180.000,B 0.000,C 180.000} C_DIS
LIN {X 109.368,Y 94.573,Z 73.500,A 180.000,B 0.000,C 180.000} C_DIS
LIN {X 109.276,Y 94.215,Z 73.500,A 180.000,B 0.000,C 180.000} C_DIS
LIN {X 109.232,Y 94.054,Z 73.500,A 180.000,B 0.000,C 180.000} C_DIS
LIN {X 109.226,Y 94.036,Z 73.500,A 180.000,B 0.000,C 180.000} C_DIS
LIN {X 109.169,Y 93.857,Z 73.500,A 180.000,B 0.000,C 180.000} C_DIS
LIN {X 109.112,Y 93.679,Z 73.500,A 180.000,B 0.000,C 180.000} C_DIS
LIN {X 109.055,Y 93.500,Z 73.500,A 180.000,B 0.000,C 180.000} C_DIS
LIN {X 109.053,Y 93.495,Z 73.500,A 180.000,B 0.000,C 180.000} C_DIS
LIN {X 108.988,Y 93.321,Z 73.500,A 180.000,B 0.000,C 180.000} C_DIS
LIN {X 108.852,Y 92.964,Z 73.500,A 180.000,B 0.000,C 180.000} C_DIS
LIN {X 108.781,Y 92.785,Z 73.500,A 180.000,B 0.000,C 180.000} C_DIS
LIN {X 108.702,Y 92.606,Z 73.500,A 180.000,B 0.000,C 180.000} C_DIS
LIN {X 108.622,Y 92.427,Z 73.500,A 180.000,B 0.000,C 180.000} C_DIS
LIN {X 108.542,Y 92.249,Z 73.500,A 180.000,B 0.000,C 180.000} C_DIS
LIN {X 108.517,Y 92.194,Z 73.500,A 180.000,B 0.000,C 180.000} C_DIS
LIN {X 108.453,Y 92.070,Z 73.500,A 180.000,B 0.000,C 180.000} C_DIS
LIN {X 108.269,Y 91.712,Z 73.500,A 180.000,B 0.000,C 180.000} C_DIS
LIN {X 108.172,Y 91.533,Z 73.500,A 180.000,B 0.000,C 180.000} C_DIS
LIN {X 108.159,Y 91.511,Z 73.500,A 180.000,B 0.000,C 180.000} C_DIS
LIN {X 108.067,Y 91.355,Z 73.500,A 180.000,B 0.000,C 180.000} C_DIS
LIN {X 107.962,Y 91.176,Z 73.500,A 180.000,B 0.000,C 180.000} C_DIS
LIN {X 107.855,Y 90.997,Z 73.500,A 180.000,B 0.000,C 180.000} C_DIS
LIN {X 107.802,Y 90.915,Z 73.500,A 180.000,B 0.000,C 180.000} C_DIS
LIN {X 107.618,Y 90.640,Z 73.500,A 180.000,B 0.000,C 180.000} C_DIS
LIN {X 107.497,Y 90.461,Z 73.500,A 180.000,B 0.000,C 180.000} C_DIS
LIN {X 107.444,Y 90.387,Z 73.500,A 180.000,B 0.000,C 180.000} C_DIS
LIN {X 107.366,Y 90.282,Z 73.500,A 180.000,B 0.000,C 180.000} C_DIS
LIN {X 107.097,Y 89.925,Z 73.500,A 180.000,B 0.000,C 180.000} C_DIS
LIN {X 107.086,Y 89.910,Z 73.500,A 180.000,B 0.000,C 180.000} C_DIS
LIN {X 106.952,Y 89.746,Z 73.500,A 180.000,B 0.000,C 180.000} C_DIS
LIN {X 106.729,Y 89.482,Z 73.500,A 180.000,B 0.000,C 180.000} C_DIS
LIN {X 106.649,Y 89.388,Z 73.500,A 180.000,B 0.000,C 180.000} C_DIS
LIN {X 106.550,Y 89.281,Z 73.500,A 180.000,B 0.000,C 180.000} C_DIS
LIN {X 106.483,Y 89.209,Z 73.500,A 180.000,B 0.000,C 180.000} C_DIS
LIN {X 106.193,Y 88.903,Z 73.500,A 180.000,B 0.000,C 180.000} C_DIS
LIN {X 106.144,Y 88.852,Z 73.500,A 180.000,B 0.000,C 180.000} C_DIS
LIN {X 106.014,Y 88.727,Z 73.500,A 180.000,B 0.000,C 180.000} C_DIS
LIN {X 105.768,Y 88.494,Z 73.500,A 180.000,B 0.000,C 180.000} C_DIS
LIN {X 105.656,Y 88.390,Z 73.500,A 180.000,B 0.000,C 180.000} C_DIS
LIN {X 105.569,Y 88.316,Z 73.500,A 180.000,B 0.000,C 180.000} C_DIS
LIN {X 105.299,Y 88.087,Z 73.500,A 180.000,B 0.000,C 180.000} C_DIS
LIN {X 105.144,Y 87.958,Z 73.500,A 180.000,B 0.000,C 180.000} C_DIS
LIN {X 105.120,Y 87.938,Z 73.500,A 180.000,B 0.000,C 180.000} C_DIS
LIN {X 104.941,Y 87.801,Z 73.500,A 180.000,B 0.000,C 180.000} C_DIS
LIN {X 104.675,Y 87.601,Z 73.500,A 180.000,B 0.000,C 180.000} C_DIS
LIN {X 104.584,Y 87.533,Z 73.500,A 180.000,B 0.000,C 180.000} C_DIS
LIN {X 104.419,Y 87.422,Z 73.500,A 180.000,B 0.000,C 180.000} C_DIS
LIN {X 104.151,Y 87.243,Z 73.500,A 180.000,B 0.000,C 180.000} C_DIS
LIN {X 104.047,Y 87.175,Z 73.500,A 180.000,B 0.000,C 180.000} C_DIS
LIN {X 103.869,Y 87.065,Z 73.500,A 180.000,B 0.000,C 180.000} C_DIS
LIN {X 103.511,Y 86.854,Z 73.500,A 180.000,B 0.000,C 180.000} C_DIS
LIN {X 103.332,Y 86.754,Z 73.500,A 180.000,B 0.000,C 180.000} C_DIS
LIN {X 102.975,Y 86.569,Z 73.500,A 180.000,B 0.000,C 180.000} C_DIS
LIN {X 102.894,Y 86.528,Z 73.500,A 180.000,B 0.000,C 180.000} C_DIS
LIN {X 102.796,Y 86.480,Z 73.500,A 180.000,B 0.000,C 180.000} C_DIS
LIN {X 102.617,Y 86.398,Z 73.500,A 180.000,B 0.000,C 180.000} C_DIS
LIN {X 102.383,Y 86.293,Z 73.500,A 180.000,B 0.000,C 180.000} C_DIS
LIN {X 102.260,Y 86.238,Z 73.500,A 180.000,B 0.000,C 180.000} C_DIS
LIN {X 102.097,Y 86.170,Z 73.500,A 180.000,B 0.000,C 180.000} C_DIS
LIN {X 101.629,Y 85.992,Z 73.500,A 180.000,B 0.000,C 180.000} C_DIS
LIN {X 101.545,Y 85.961,Z 73.500,A 180.000,B 0.000,C 180.000} C_DIS
LIN {X 101.366,Y 85.903,Z 73.500,A 180.000,B 0.000,C 180.000} C_DIS
LIN {X 101.008,Y 85.789,Z 73.500,A 180.000,B 0.000,C 180.000} C_DIS
LIN {X 100.829,Y 85.735,Z 73.500,A 180.000,B 0.000,C 180.000} C_DIS
LIN {X 100.651,Y 85.688,Z 73.500,A 180.000,B 0.000,C 180.000} C_DIS
LIN {X 100.440,Y 85.634,Z 73.500,A 180.000,B 0.000,C 180.000} C_DIS
LIN {X 100.293,Y 85.596,Z 73.500,A 180.000,B 0.000,C 180.000} C_DIS
LIN {X 100.114,Y 85.557,Z 73.500,A 180.000,B 0.000,C 180.000} C_DIS
LIN {X 99.757,Y 85.486,Z 73.500,A 180.000,B 0.000,C 180.000} C_DIS
LIN {X 99.598,Y 85.455,Z 73.500,A 180.000,B 0.000,C 180.000} C_DIS
LIN {X 99.578,Y 85.451,Z 73.500,A 180.000,B 0.000,C 180.000} C_DIS
LIN {X 99.399,Y 85.423,Z 73.500,A 180.000,B 0.000,C 180.000} C_DIS
LIN {X 99.042,Y 85.372,Z 73.500,A 180.000,B 0.000,C 180.000} C_DIS
LIN {X 98.863,Y 85.349,Z 73.500,A 180.000,B 0.000,C 180.000} C_DIS
LIN {X 98.684,Y 85.333,Z 73.500,A 180.000,B 0.000,C 180.000} C_DIS
LIN {X 98.327,Y 85.303,Z 73.500,A 180.000,B 0.000,C 180.000} C_DIS
LIN {X 98.148,Y 85.290,Z 73.500,A 180.000,B 0.000,C 180.000} C_DIS
LIN {X 97.969,Y 85.284,Z 73.500,A 180.000,B 0.000,C 180.000} C_DIS
LIN {X 97.612,Y 85.274,Z 73.500,A 180.000,B 0.000,C 180.000} C_DIS
LIN {X 97.433,Y 85.273,Z 73.500,A 180.000,B 0.000,C 180.000} C_DIS
LIN {X 97.075,Y 85.283,Z 73.500,A 180.000,B 0.000,C 180.000} C_DIS
LIN {X 96.897,Y 85.288,Z 73.500,A 180.000,B 0.000,C 180.000} C_DIS
LIN {X 96.718,Y 85.299,Z 73.500,A 180.000,B 0.000,C 180.000} C_DIS
LIN {X 96.539,Y 85.314,Z 73.500,A 180.000,B 0.000,C 180.000} C_DIS
LIN {X 96.360,Y 85.329,Z 73.500,A 180.000,B 0.000,C 180.000} C_DIS
LIN {X 96.181,Y 85.344,Z 73.500,A 180.000,B 0.000,C 180.000} C_DIS
LIN {X 96.003,Y 85.366,Z 73.500,A 180.000,B 0.000,C 180.000} C_DIS
LIN {X 95.645,Y 85.417,Z 73.500,A 180.000,B 0.000,C 180.000} C_DIS
LIN {X 95.466,Y 85.443,Z 73.500,A 180.000,B 0.000,C 180.000} C_DIS
LIN {X 95.402,Y 85.455,Z 73.500,A 180.000,B 0.000,C 180.000} C_DIS
LIN {X 95.288,Y 85.477,Z 73.500,A 180.000,B 0.000,C 180.000} C_DIS
LIN {X 94.930,Y 85.549,Z 73.500,A 180.000,B 0.000,C 180.000} C_DIS
LIN {X 94.751,Y 85.585,Z 73.500,A 180.000,B 0.000,C 180.000} C_DIS
LIN {X 94.573,Y 85.631,Z 73.500,A 180.000,B 0.000,C 180.000} C_DIS
LIN {X 94.215,Y 85.723,Z 73.500,A 180.000,B 0.000,C 180.000} C_DIS
LIN {X 94.036,Y 85.775,Z 73.500,A 180.000,B 0.000,C 180.000} C_DIS
LIN {X 93.679,Y 85.889,Z 73.500,A 180.000,B 0.000,C 180.000} C_DIS
LIN {X 93.500,Y 85.947,Z 73.500,A 180.000,B 0.000,C 180.000} C_DIS
LIN {X 93.371,Y 85.992,Z 73.500,A 180.000,B 0.000,C 180.000} C_DIS
LIN {X 92.903,Y 86.170,Z 73.500,A 180.000,B 0.000,C 180.000} C_DIS
LIN {X 92.785,Y 86.218,Z 73.500,A 180.000,B 0.000,C 180.000} C_DIS
LIN {X 92.606,Y 86.298,Z 73.500,A 180.000,B 0.000,C 180.000} C_DIS
LIN {X 92.427,Y 86.378,Z 73.500,A 180.000,B 0.000,C 180.000} C_DIS
LIN {X 92.249,Y 86.459,Z 73.500,A 180.000,B 0.000,C 180.000} C_DIS
LIN {X 92.106,Y 86.528,Z 73.500,A 180.000,B 0.000,C 180.000} C_DIS
LIN {X 92.070,Y 86.546,Z 73.500,A 180.000,B 0.000,C 180.000} C_DIS
LIN {X 91.712,Y 86.731,Z 73.500,A 180.000,B 0.000,C 180.000} C_DIS
LIN {X 91.533,Y 86.827,Z 73.500,A 180.000,B 0.000,C 180.000} C_DIS
LIN {X 91.435,Y 86.885,Z 73.500,A 180.000,B 0.000,C 180.000} C_DIS
LIN {X 91.132,Y 87.064,Z 73.500,A 180.000,B 0.000,C 180.000} C_DIS
LIN {X 90.997,Y 87.146,Z 73.500,A 180.000,B 0.000,C 180.000} C_DIS
LIN {X 90.849,Y 87.243,Z 73.500,A 180.000,B 0.000,C 180.000} C_DIS
LIN {X 90.581,Y 87.422,Z 73.500,A 180.000,B 0.000,C 180.000} C_DIS
LIN {X 90.461,Y 87.502,Z 73.500,A 180.000,B 0.000,C 180.000} C_DIS
LIN {X 90.325,Y 87.601,Z 73.500,A 180.000,B 0.000,C 180.000} C_DIS
LIN {X 90.088,Y 87.779,Z 73.500,A 180.000,B 0.000,C 180.000} C_DIS
LIN {X 89.925,Y 87.902,Z 73.500,A 180.000,B 0.000,C 180.000} C_DIS
LIN {X 89.856,Y 87.958,Z 73.500,A 180.000,B 0.000,C 180.000} C_DIS
LIN {X 89.746,Y 88.050,Z 73.500,A 180.000,B 0.000,C 180.000} C_DIS
LIN {X 89.431,Y 88.316,Z 73.500,A 180.000,B 0.000,C 180.000} C_DIS
LIN {X 89.388,Y 88.352,Z 73.500,A 180.000,B 0.000,C 180.000} C_DIS
LIN {X 89.232,Y 88.494,Z 73.500,A 180.000,B 0.000,C 180.000} C_DIS
LIN {X 89.031,Y 88.685,Z 73.500,A 180.000,B 0.000,C 180.000} C_DIS
LIN {X 88.856,Y 88.852,Z 73.500,A 180.000,B 0.000,C 180.000} C_DIS
LIN {X 88.852,Y 88.856,Z 73.500,A 180.000,B 0.000,C 180.000} C_DIS
LIN {X 88.686,Y 89.031,Z 73.500,A 180.000,B 0.000,C 180.000} C_DIS
LIN {X 88.494,Y 89.234,Z 73.500,A 180.000,B 0.000,C 180.000} C_DIS
LIN {X 88.351,Y 89.388,Z 73.500,A 180.000,B 0.000,C 180.000} C_DIS
LIN {X 88.316,Y 89.429,Z 73.500,A 180.000,B 0.000,C 180.000} C_DIS
LIN {X 88.048,Y 89.746,Z 73.500,A 180.000,B 0.000,C 180.000} C_DIS
LIN {X 87.958,Y 89.854,Z 73.500,A 180.000,B 0.000,C 180.000} C_DIS
LIN {X 87.903,Y 89.925,Z 73.500,A 180.000,B 0.000,C 180.000} C_DIS
LIN {X 87.601,Y 90.326,Z 73.500,A 180.000,B 0.000,C 180.000} C_DIS
LIN {X 87.503,Y 90.461,Z 73.500,A 180.000,B 0.000,C 180.000} C_DIS
LIN {X 87.422,Y 90.581,Z 73.500,A 180.000,B 0.000,C 180.000} C_DIS
LIN {X 87.243,Y 90.848,Z 73.500,A 180.000,B 0.000,C 180.000} C_DIS
LIN {X 87.145,Y 90.997,Z 73.500,A 180.000,B 0.000,C 180.000} C_DIS
LIN {X 87.064,Y 91.132,Z 73.500,A 180.000,B 0.000,C 180.000} C_DIS
LIN {X 86.885,Y 91.435,Z 73.500,A 180.000,B 0.000,C 180.000} C_DIS
LIN {X 86.828,Y 91.533,Z 73.500,A 180.000,B 0.000,C 180.000} C_DIS
LIN {X 86.731,Y 91.712,Z 73.500,A 180.000,B 0.000,C 180.000} C_DIS
LIN {X 86.528,Y 92.106,Z 73.500,A 180.000,B 0.000,C 180.000} C_DIS
LIN {X 86.458,Y 92.249,Z 73.500,A 180.000,B 0.000,C 180.000} C_DIS
LIN {X 86.378,Y 92.427,Z 73.500,A 180.000,B 0.000,C 180.000} C_DIS
LIN {X 86.298,Y 92.606,Z 73.500,A 180.000,B 0.000,C 180.000} C_DIS
LIN {X 86.219,Y 92.785,Z 73.500,A 180.000,B 0.000,C 180.000} C_DIS
LIN {X 86.170,Y 92.906,Z 73.500,A 180.000,B 0.000,C 180.000} C_DIS
LIN {X 86.148,Y 92.964,Z 73.500,A 180.000,B 0.000,C 180.000} C_DIS
LIN {X 85.992,Y 93.374,Z 73.500,A 180.000,B 0.000,C 180.000} C_DIS
LIN {X 85.945,Y 93.500,Z 73.500,A 180.000,B 0.000,C 180.000} C_DIS
LIN {X 85.888,Y 93.679,Z 73.500,A 180.000,B 0.000,C 180.000} C_DIS
LIN {X 85.813,Y 93.914,Z 73.500,A 180.000,B 0.000,C 180.000} C_DIS
LIN {X 85.774,Y 94.036,Z 73.500,A 180.000,B 0.000,C 180.000} C_DIS
LIN {X 85.724,Y 94.215,Z 73.500,A 180.000,B 0.000,C 180.000} C_DIS
LIN {X 85.632,Y 94.573,Z 73.500,A 180.000,B 0.000,C 180.000} C_DIS
LIN {X 85.586,Y 94.751,Z 73.500,A 180.000,B 0.000,C 180.000} C_DIS
LIN {X 85.548,Y 94.930,Z 73.500,A 180.000,B 0.000,C 180.000} C_DIS
LIN {X 85.476,Y 95.288,Z 73.500,A 180.000,B 0.000,C 180.000} C_DIS
LIN {X 85.455,Y 95.395,Z 73.500,A 180.000,B 0.000,C 180.000} C_DIS
LIN {X 85.443,Y 95.466,Z 73.500,A 180.000,B 0.000,C 180.000} C_DIS
LIN {X 85.417,Y 95.645,Z 73.500,A 180.000,B 0.000,C 180.000} C_DIS
LIN {X 85.367,Y 96.003,Z 73.500,A 180.000,B 0.000,C 180.000} C_DIS
LIN {X 85.344,Y 96.181,Z 73.500,A 180.000,B 0.000,C 180.000} C_DIS
LIN {X 85.329,Y 96.360,Z 73.500,A 180.000,B 0.000,C 180.000} C_DIS
LIN {X 85.299,Y 96.718,Z 73.500,A 180.000,B 0.000,C 180.000} C_DIS
LIN {X 85.288,Y 96.897,Z 73.500,A 180.000,B 0.000,C 180.000} C_DIS
LIN {X 85.276,Y 97.318,Z 73.500,A 180.000,B 0.000,C 180.000} C_DIS
LIN {X 85.274,Y 97.433,Z 73.500,A 180.000,B 0.000,C 180.000} C_DIS
LIN {X 85.275,Y 97.612,Z 73.500,A 180.000,B 0.000,C 180.000} C_DIS
LIN {X 85.285,Y 97.969,Z 73.500,A 180.000,B 0.000,C 180.000} C_DIS
LIN {X 85.290,Y 98.148,Z 73.500,A 180.000,B 0.000,C 180.000} C_DIS
LIN {X 85.302,Y 98.327,Z 73.500,A 180.000,B 0.000,C 180.000} C_DIS
LIN {X 85.332,Y 98.684,Z 73.500,A 180.000,B 0.000,C 180.000} C_DIS
LIN {X 85.349,Y 98.863,Z 73.500,A 180.000,B 0.000,C 180.000} C_DIS
LIN {X 85.373,Y 99.042,Z 73.500,A 180.000,B 0.000,C 180.000} C_DIS
LIN {X 85.424,Y 99.399,Z 73.500,A 180.000,B 0.000,C 180.000} C_DIS
LIN {X 85.450,Y 99.578,Z 73.500,A 180.000,B 0.000,C 180.000} C_DIS
LIN {X 85.455,Y 99.605,Z 73.500,A 180.000,B 0.000,C 180.000} C_DIS
LIN {X 85.485,Y 99.757,Z 73.500,A 180.000,B 0.000,C 180.000} C_DIS
LIN {X 85.556,Y 100.114,Z 73.500,A 180.000,B 0.000,C 180.000} C_DIS
LIN {X 85.598,Y 100.293,Z 73.500,A 180.000,B 0.000,C 180.000} C_DIS
LIN {X 85.634,Y 100.435,Z 73.500,A 180.000,B 0.000,C 180.000} C_DIS
LIN {X 85.736,Y 100.829,Z 73.500,A 180.000,B 0.000,C 180.000} C_DIS
LIN {X 85.788,Y 101.008,Z 73.500,A 180.000,B 0.000,C 180.000} C_DIS
LIN {X 85.902,Y 101.366,Z 73.500,A 180.000,B 0.000,C 180.000} C_DIS
LIN {X 85.961,Y 101.545,Z 73.500,A 180.000,B 0.000,C 180.000} C_DIS
LIN {X 85.992,Y 101.626,Z 73.500,A 180.000,B 0.000,C 180.000} C_DIS
LIN {X 86.097,Y 101.902,Z 73.500,A 180.000,B 0.000,C 180.000} C_DIS
LIN {X 86.165,Y 102.081,Z 73.500,A 180.000,B 0.000,C 180.000} C_DIS
LIN {X 86.170,Y 102.094,Z 73.500,A 180.000,B 0.000,C 180.000} C_DIS
LIN {X 86.238,Y 102.260,Z 73.500,A 180.000,B 0.000,C 180.000} C_DIS
LIN {X 86.318,Y 102.438,Z 73.500,A 180.000,B 0.000,C 180.000} C_DIS
LIN {X 86.398,Y 102.617,Z 73.500,A 180.000,B 0.000,C 180.000} C_DIS
LIN {X 86.479,Y 102.796,Z 73.500,A 180.000,B 0.000,C 180.000} C_DIS
LIN {X 86.528,Y 102.894,Z 73.500,A 180.000,B 0.000,C 180.000} C_DIS
LIN {X 86.707,Y 103.240,Z 73.500,A 180.000,B 0.000,C 180.000} C_DIS
LIN {X 86.755,Y 103.332,Z 73.500,A 180.000,B 0.000,C 180.000} C_DIS
LIN {X 86.854,Y 103.511,Z 73.500,A 180.000,B 0.000,C 180.000} C_DIS
LIN {X 87.065,Y 103.869,Z 73.500,A 180.000,B 0.000,C 180.000} C_DIS
LIN {X 87.173,Y 104.047,Z 73.500,A 180.000,B 0.000,C 180.000} C_DIS
LIN {X 87.243,Y 104.152,Z 73.500,A 180.000,B 0.000,C 180.000} C_DIS
LIN {X 87.422,Y 104.419,Z 73.500,A 180.000,B 0.000,C 180.000} C_DIS
LIN {X 87.535,Y 104.584,Z 73.500,A 180.000,B 0.000,C 180.000} C_DIS
LIN {X 87.601,Y 104.674,Z 73.500,A 180.000,B 0.000,C 180.000} C_DIS
LIN {X 87.802,Y 104.941,Z 73.500,A 180.000,B 0.000,C 180.000} C_DIS
LIN {X 87.937,Y 105.120,Z 73.500,A 180.000,B 0.000,C 180.000} C_DIS
LIN {X 87.958,Y 105.146,Z 73.500,A 180.000,B 0.000,C 180.000} C_DIS
LIN {X 88.086,Y 105.299,Z 73.500,A 180.000,B 0.000,C 180.000} C_DIS
LIN {X 88.316,Y 105.571,Z 73.500,A 180.000,B 0.000,C 180.000} C_DIS
LIN {X 88.391,Y 105.656,Z 73.500,A 180.000,B 0.000,C 180.000} C_DIS
LIN {X 88.494,Y 105.766,Z 73.500,A 180.000,B 0.000,C 180.000} C_DIS
LIN {X 88.728,Y 106.014,Z 73.500,A 180.000,B 0.000,C 180.000} C_DIS
LIN {X 88.852,Y 106.144,Z 73.500,A 180.000,B 0.000,C 180.000} C_DIS
LIN {X 88.901,Y 106.193,Z 73.500,A 180.000,B 0.000,C 180.000} C_DIS
LIN {X 89.031,Y 106.315,Z 73.500,A 180.000,B 0.000,C 180.000} C_DIS
LIN {X 89.279,Y 106.550,Z 73.500,A 180.000,B 0.000,C 180.000} C_DIS
LIN {X 89.388,Y 106.648,Z 73.500,A 180.000,B 0.000,C 180.000} C_DIS
LIN {X 89.746,Y 106.950,Z 73.500,A 180.000,B 0.000,C 180.000} C_DIS
LIN {X 89.910,Y 107.086,Z 73.500,A 180.000,B 0.000,C 180.000} C_DIS
LIN {X 89.925,Y 107.098,Z 73.500,A 180.000,B 0.000,C 180.000} C_DIS
LIN {X 90.103,Y 107.232,Z 73.500,A 180.000,B 0.000,C 180.000} C_DIS
LIN {X 90.282,Y 107.367,Z 73.500,A 180.000,B 0.000,C 180.000} C_DIS
LIN {X 90.385,Y 107.444,Z 73.500,A 180.000,B 0.000,C 180.000} C_DIS
LIN {X 90.461,Y 107.498,Z 73.500,A 180.000,B 0.000,C 180.000} C_DIS
LIN {X 90.648,Y 107.623,Z 73.500,A 180.000,B 0.000,C 180.000} C_DIS
LIN {X 90.818,Y 107.737,Z 73.500,A 180.000,B 0.000,C 180.000} C_DIS
LIN {X 90.915,Y 107.802,Z 73.500,A 180.000,B 0.000,C 180.000} C_DIS
LIN {X 90.997,Y 107.854,Z 73.500,A 180.000,B 0.000,C 180.000} C_DIS
LIN {X 91.176,Y 107.962,Z 73.500,A 180.000,B 0.000,C 180.000} C_DIS
LIN {X 91.510,Y 108.159,Z 73.500,A 180.000,B 0.000,C 180.000} C_DIS
LIN {X 91.533,Y 108.173,Z 73.500,A 180.000,B 0.000,C 180.000} C_DIS
LIN {X 91.712,Y 108.269,Z 73.500,A 180.000,B 0.000,C 180.000} C_DIS
LIN {X 92.070,Y 108.454,Z 73.500,A 180.000,B 0.000,C 180.000} C_DIS
LIN {X 92.082,Y 108.460,Z 73.500,A 180.000,B 0.000,C 180.000} C_DIS
; Link Move Starts
LIN {X 92.343,Y 108.584,Z 73.500,A 180.000,B 0.000,C 180.000} C_DIS
LIN {X 92.630,Y 108.713,Z 73.499,A 180.000,B 0.000,C 180.000} C_DIS
LIN {X 92.898,Y 108.829,Z 73.498,A 180.000,B 0.000,C 180.000} C_DIS
LIN {X 93.189,Y 108.941,Z 73.496,A 180.000,B 0.000,C 180.000} C_DIS
LIN {X 93.472,Y 109.047,Z 73.494,A 180.000,B 0.000,C 180.000} C_DIS
LIN {X 93.759,Y 109.140,Z 73.492,A 180.000,B 0.000,C 180.000} C_DIS
LIN {X 94.053,Y 109.236,Z 73.489,A 180.000,B 0.000,C 180.000} C_DIS
LIN {X 94.337,Y 109.315,Z 73.486,A 180.000,B 0.000,C 180.000} C_DIS
LIN {X 94.642,Y 109.396,Z 73.482,A 180.000,B 0.000,C 180.000} C_DIS
LIN {X 94.924,Y 109.460,Z 73.478,A 180.000,B 0.000,C 180.000} C_DIS
LIN {X 95.232,Y 109.524,Z 73.474,A 180.000,B 0.000,C 180.000} C_DIS
LIN {X 95.531,Y 109.582,Z 73.469,A 180.000,B 0.000,C 180.000} C_DIS
LIN {X 95.679,Y 109.604,Z 73.467,A 180.000,B 0.000,C 180.000} C_DIS
LIN {X 95.828,Y 109.626,Z 73.464,A 180.000,B 0.000,C 180.000} C_DIS
LIN {X 95.976,Y 109.648,Z 73.461,A 180.000,B 0.000,C 180.000} C_DIS
LIN {X 96.124,Y 109.669,Z 73.459,A 180.000,B 0.000,C 180.000} C_DIS
LIN {X 96.276,Y 109.685,Z 73.456,A 180.000,B 0.000,C 180.000} C_DIS
LIN {X 96.428,Y 109.699,Z 73.453,A 180.000,B 0.000,C 180.000} C_DIS
LIN {X 96.585,Y 109.713,Z 73.450,A 180.000,B 0.000,C 180.000} C_DIS
LIN {X 96.741,Y 109.728,Z 73.446,A 180.000,B 0.000,C 180.000} C_DIS
LIN {X 96.886,Y 109.738,Z 73.443,A 180.000,B 0.000,C 180.000} C_DIS
LIN {X 97.032,Y 109.744,Z 73.440,A 180.000,B 0.000,C 180.000} C_DIS
LIN {X 97.189,Y 109.750,Z 73.437,A 180.000,B 0.000,C 180.000} C_DIS
LIN {X 97.347,Y 109.756,Z 73.433,A 180.000,B 0.000,C 180.000} C_DIS
LIN {X 97.492,Y 109.761,Z 73.430,A 180.000,B 0.000,C 180.000} C_DIS
LIN {X 97.637,Y 109.759,Z 73.426,A 180.000,B 0.000,C 180.000} C_DIS
LIN {X 97.795,Y 109.757,Z 73.422,A 180.000,B 0.000,C 180.000} C_DIS
LIN {X 97.952,Y 109.754,Z 73.418,A 180.000,B 0.000,C 180.000} C_DIS
LIN {X 98.102,Y 109.752,Z 73.415,A 180.000,B 0.000,C 180.000} C_DIS
LIN {X 98.252,Y 109.745,Z 73.411,A 180.000,B 0.000,C 180.000} C_DIS
LIN {X 98.405,Y 109.734,Z 73.407,A 180.000,B 0.000,C 180.000} C_DIS
LIN {X 98.557,Y 109.723,Z 73.403,A 180.000,B 0.000,C 180.000} C_DIS
LIN {X 98.707,Y 109.713,Z 73.398,A 180.000,B 0.000,C 180.000} C_DIS
LIN {X 98.857,Y 109.702,Z 73.394,A 180.000,B 0.000,C 180.000} C_DIS
LIN {X 99.009,Y 109.684,Z 73.390,A 180.000,B 0.000,C 180.000} C_DIS
LIN {X 99.161,Y 109.665,Z 73.386,A 180.000,B 0.000,C 180.000} C_DIS
LIN {X 99.317,Y 109.645,Z 73.381,A 180.000,B 0.000,C 180.000} C_DIS
LIN {X 99.473,Y 109.625,Z 73.376,A 180.000,B 0.000,C 180.000} C_DIS
LIN {X 99.617,Y 109.602,Z 73.372,A 180.000,B 0.000,C 180.000} C_DIS
LIN {X 99.762,Y 109.576,Z 73.367,A 180.000,B 0.000,C 180.000} C_DIS
LIN {X 99.916,Y 109.547,Z 73.363,A 180.000,B 0.000,C 180.000} C_DIS
LIN {X 100.071,Y 109.519,Z 73.358,A 180.000,B 0.000,C 180.000} C_DIS
LIN {X 100.218,Y 109.492,Z 73.353,A 180.000,B 0.000,C 180.000} C_DIS
LIN {X 100.364,Y 109.459,Z 73.348,A 180.000,B 0.000,C 180.000} C_DIS
LIN {X 100.439,Y 109.441,Z 73.346,A 180.000,B 0.000,C 180.000} C_DIS
LIN {X 100.514,Y 109.422,Z 73.343,A 180.000,B 0.000,C 180.000} C_DIS
LIN {X 100.589,Y 109.404,Z 73.341,A 180.000,B 0.000,C 180.000} C_DIS
LIN {X 100.664,Y 109.386,Z 73.338,A 180.000,B 0.000,C 180.000} C_DIS
LIN {X 100.808,Y 109.351,Z 73.333,A 180.000,B 0.000,C 180.000} C_DIS
LIN {X 100.950,Y 109.313,Z 73.328,A 180.000,B 0.000,C 180.000} C_DIS
LIN {X 101.100,Y 109.268,Z 73.323,A 180.000,B 0.000,C 180.000} C_DIS
LIN {X 101.175,Y 109.246,Z 73.320,A 180.000,B 0.000,C 180.000} C_DIS
LIN {X 101.250,Y 109.223,Z 73.318,A 180.000,B 0.000,C 180.000} C_DIS
LIN {X 101.325,Y 109.200,Z 73.315,A 180.000,B 0.000,C 180.000} C_DIS
LIN {X 101.399,Y 109.178,Z 73.312,A 180.000,B 0.000,C 180.000} C_DIS
LIN {X 101.474,Y 109.155,Z 73.309,A 180.000,B 0.000,C 180.000} C_DIS
LIN {X 101.549,Y 109.133,Z 73.307,A 180.000,B 0.000,C 180.000} C_DIS
LIN {X 101.619,Y 109.109,Z 73.304,A 180.000,B 0.000,C 180.000} C_DIS
LIN {X 101.689,Y 109.084,Z 73.302,A 180.000,B 0.000,C 180.000} C_DIS
LIN {X 101.903,Y 109.007,Z 73.294,A 180.000,B 0.000,C 180.000} C_DIS
LIN {X 102.051,Y 108.953,Z 73.288,A 180.000,B 0.000,C 180.000} C_DIS
LIN {X 102.125,Y 108.926,Z 73.285,A 180.000,B 0.000,C 180.000} C_DIS
LIN {X 102.194,Y 108.900,Z 73.283,A 180.000,B 0.000,C 180.000} C_DIS
LIN {X 102.262,Y 108.873,Z 73.280,A 180.000,B 0.000,C 180.000} C_DIS
LIN {X 102.330,Y 108.844,Z 73.278,A 180.000,B 0.000,C 180.000} C_DIS
LIN {X 102.398,Y 108.815,Z 73.275,A 180.000,B 0.000,C 180.000} C_DIS
LIN {X 102.542,Y 108.753,Z 73.270,A 180.000,B 0.000,C 180.000} C_DIS
LIN {X 102.686,Y 108.692,Z 73.264,A 180.000,B 0.000,C 180.000} C_DIS
LIN {X 102.755,Y 108.662,Z 73.262,A 180.000,B 0.000,C 180.000} C_DIS
LIN {X 102.825,Y 108.631,Z 73.259,A 180.000,B 0.000,C 180.000} C_DIS
LIN {X 102.894,Y 108.599,Z 73.256,A 180.000,B 0.000,C 180.000} C_DIS
LIN {X 102.962,Y 108.566,Z 73.254,A 180.000,B 0.000,C 180.000} C_DIS
LIN {X 103.100,Y 108.498,Z 73.248,A 180.000,B 0.000,C 180.000} C_DIS
LIN {X 103.308,Y 108.395,Z 73.240,A 180.000,B 0.000,C 180.000} C_DIS
LIN {X 103.377,Y 108.360,Z 73.237,A 180.000,B 0.000,C 180.000} C_DIS
LIN {X 103.446,Y 108.326,Z 73.235,A 180.000,B 0.000,C 180.000} C_DIS
LIN {X 103.515,Y 108.289,Z 73.232,A 180.000,B 0.000,C 180.000} C_DIS
LIN {X 103.580,Y 108.252,Z 73.229,A 180.000,B 0.000,C 180.000} C_DIS
LIN {X 103.711,Y 108.178,Z 73.224,A 180.000,B 0.000,C 180.000} C_DIS
LIN {X 103.777,Y 108.140,Z 73.221,A 180.000,B 0.000,C 180.000} C_DIS
LIN {X 103.913,Y 108.063,Z 73.216,A 180.000,B 0.000,C 180.000} C_DIS
LIN {X 103.981,Y 108.025,Z 73.213,A 180.000,B 0.000,C 180.000} C_DIS
LIN {X 104.048,Y 107.985,Z 73.211,A 180.000,B 0.000,C 180.000} C_DIS
LIN {X 104.112,Y 107.946,Z 73.208,A 180.000,B 0.000,C 180.000} C_DIS
LIN {X 104.175,Y 107.906,Z 73.205,A 180.000,B 0.000,C 180.000} C_DIS
LIN {X 104.565,Y 107.655,Z 73.189,A 180.000,B 0.000,C 180.000} C_DIS
LIN {X 104.628,Y 107.614,Z 73.186,A 180.000,B 0.000,C 180.000} C_DIS
LIN {X 104.689,Y 107.573,Z 73.184,A 180.000,B 0.000,C 180.000} C_DIS
LIN {X 104.750,Y 107.529,Z 73.181,A 180.000,B 0.000,C 180.000} C_DIS
LIN {X 104.810,Y 107.485,Z 73.179,A 180.000,B 0.000,C 180.000} C_DIS
LIN {X 104.937,Y 107.393,Z 73.173,A 180.000,B 0.000,C 180.000} C_DIS
LIN {X 105.125,Y 107.256,Z 73.165,A 180.000,B 0.000,C 180.000} C_DIS
LIN {X 105.185,Y 107.212,Z 73.163,A 180.000,B 0.000,C 180.000} C_DIS
LIN {X 105.243,Y 107.166,Z 73.160,A 180.000,B 0.000,C 180.000} C_DIS
LIN {X 105.301,Y 107.119,Z 73.157,A 180.000,B 0.000,C 180.000} C_DIS
LIN {X 105.362,Y 107.070,Z 73.155,A 180.000,B 0.000,C 180.000} C_DIS
LIN {X 105.666,Y 106.822,Z 73.141,A 180.000,B 0.000,C 180.000} C_DIS
LIN {X 105.726,Y 106.773,Z 73.138,A 180.000,B 0.000,C 180.000} C_DIS
LIN {X 105.785,Y 106.723,Z 73.135,A 180.000,B 0.000,C 180.000} C_DIS
LIN {X 105.841,Y 106.672,Z 73.133,A 180.000,B 0.000,C 180.000} C_DIS
LIN {X 106.178,Y 106.364,Z 73.117,A 180.000,B 0.000,C 180.000} C_DIS
LIN {X 106.234,Y 106.312,Z 73.114,A 180.000,B 0.000,C 180.000} C_DIS
LIN {X 106.289,Y 106.259,Z 73.112,A 180.000,B 0.000,C 180.000} C_DIS
LIN {X 106.343,Y 106.204,Z 73.109,A 180.000,B 0.000,C 180.000} C_DIS
LIN {X 106.671,Y 105.868,Z 73.092,A 180.000,B 0.000,C 180.000} C_DIS
LIN {X 106.723,Y 105.814,Z 73.090,A 180.000,B 0.000,C 180.000} C_DIS
LIN {X 106.775,Y 105.760,Z 73.087,A 180.000,B 0.000,C 180.000} C_DIS
LIN {X 106.825,Y 105.704,Z 73.085,A 180.000,B 0.000,C 180.000} C_DIS
LIN {X 107.082,Y 105.410,Z 73.071,A 180.000,B 0.000,C 180.000} C_DIS
LIN {X 107.131,Y 105.354,Z 73.068,A 180.000,B 0.000,C 180.000} C_DIS
LIN {X 107.180,Y 105.297,Z 73.066,A 180.000,B 0.000,C 180.000} C_DIS
LIN {X 107.228,Y 105.239,Z 73.063,A 180.000,B 0.000,C 180.000} C_DIS
LIN {X 107.275,Y 105.180,Z 73.060,A 180.000,B 0.000,C 180.000} C_DIS
LIN {X 107.563,Y 104.810,Z 73.044,A 180.000,B 0.000,C 180.000} C_DIS
LIN {X 107.610,Y 104.749,Z 73.041,A 180.000,B 0.000,C 180.000} C_DIS
LIN {X 107.656,Y 104.687,Z 73.039,A 180.000,B 0.000,C 180.000} C_DIS
LIN {X 107.701,Y 104.625,Z 73.036,A 180.000,B 0.000,C 180.000} C_DIS
LIN {X 107.745,Y 104.562,Z 73.033,A 180.000,B 0.000,C 180.000} C_DIS
LIN {X 107.966,Y 104.243,Z 73.020,A 180.000,B 0.000,C 180.000} C_DIS
LIN {X 108.010,Y 104.178,Z 73.017,A 180.000,B 0.000,C 180.000} C_DIS
LIN {X 108.052,Y 104.115,Z 73.014,A 180.000,B 0.000,C 180.000} C_DIS
LIN {X 108.092,Y 104.050,Z 73.012,A 180.000,B 0.000,C 180.000} C_DIS
LIN {X 108.336,Y 103.653,Z 72.995,A 180.000,B 0.000,C 180.000} C_DIS
LIN {X 108.375,Y 103.588,Z 72.993,A 180.000,B 0.000,C 180.000} C_DIS
LIN {X 108.413,Y 103.522,Z 72.990,A 180.000,B 0.000,C 180.000} C_DIS
LIN {X 108.450,Y 103.456,Z 72.988,A 180.000,B 0.000,C 180.000} C_DIS
LIN {X 108.486,Y 103.390,Z 72.985,A 180.000,B 0.000,C 180.000} C_DIS
LIN {X 108.707,Y 102.979,Z 72.969,A 180.000,B 0.000,C 180.000} C_DIS
LIN {X 108.742,Y 102.911,Z 72.966,A 180.000,B 0.000,C 180.000} C_DIS
LIN {X 108.775,Y 102.843,Z 72.963,A 180.000,B 0.000,C 180.000} C_DIS
LIN {X 108.974,Y 102.418,Z 72.947,A 180.000,B 0.000,C 180.000} C_DIS
LIN {X 109.007,Y 102.347,Z 72.944,A 180.000,B 0.000,C 180.000} C_DIS
LIN {X 109.038,Y 102.276,Z 72.941,A 180.000,B 0.000,C 180.000} C_DIS
LIN {X 109.067,Y 102.205,Z 72.939,A 180.000,B 0.000,C 180.000} C_DIS
LIN {X 109.096,Y 102.134,Z 72.936,A 180.000,B 0.000,C 180.000} C_DIS
LIN {X 109.271,Y 101.698,Z 72.920,A 180.000,B 0.000,C 180.000} C_DIS
LIN {X 109.298,Y 101.627,Z 72.917,A 180.000,B 0.000,C 180.000} C_DIS
LIN {X 109.324,Y 101.556,Z 72.914,A 180.000,B 0.000,C 180.000} C_DIS
LIN {X 109.372,Y 101.411,Z 72.909,A 180.000,B 0.000,C 180.000} C_DIS
LIN {X 109.447,Y 101.189,Z 72.901,A 180.000,B 0.000,C 180.000} C_DIS
LIN {X 109.497,Y 101.042,Z 72.895,A 180.000,B 0.000,C 180.000} C_DIS
LIN {X 109.520,Y 100.969,Z 72.893,A 180.000,B 0.000,C 180.000} C_DIS
LIN {X 109.541,Y 100.895,Z 72.890,A 180.000,B 0.000,C 180.000} C_DIS
LIN {X 109.582,Y 100.745,Z 72.885,A 180.000,B 0.000,C 180.000} C_DIS
LIN {X 109.665,Y 100.444,Z 72.874,A 180.000,B 0.000,C 180.000} C_DIS
LIN {X 109.686,Y 100.370,Z 72.871,A 180.000,B 0.000,C 180.000} C_DIS
LIN {X 109.706,Y 100.296,Z 72.868,A 180.000,B 0.000,C 180.000} C_DIS
LIN {X 109.724,Y 100.222,Z 72.866,A 180.000,B 0.000,C 180.000} C_DIS
LIN {X 109.740,Y 100.145,Z 72.863,A 180.000,B 0.000,C 180.000} C_DIS
LIN {X 109.839,Y 99.686,Z 72.847,A 180.000,B 0.000,C 180.000} C_DIS
LIN {X 109.855,Y 99.609,Z 72.844,A 180.000,B 0.000,C 180.000} C_DIS
LIN {X 109.868,Y 99.533,Z 72.841,A 180.000,B 0.000,C 180.000} C_DIS
LIN {X 109.892,Y 99.380,Z 72.836,A 180.000,B 0.000,C 180.000} C_DIS
LIN {X 109.904,Y 99.304,Z 72.833,A 180.000,B 0.000,C 180.000} C_DIS
LIN {X 109.928,Y 99.150,Z 72.828,A 180.000,B 0.000,C 180.000} C_DIS
LIN {X 109.940,Y 99.073,Z 72.825,A 180.000,B 0.000,C 180.000} C_DIS
LIN {X 109.953,Y 98.995,Z 72.822,A 180.000,B 0.000,C 180.000} C_DIS
LIN {X 109.963,Y 98.919,Z 72.819,A 180.000,B 0.000,C 180.000} C_DIS
LIN {X 109.974,Y 98.842,Z 72.817,A 180.000,B 0.000,C 180.000} C_DIS
LIN {X 109.982,Y 98.765,Z 72.814,A 180.000,B 0.000,C 180.000} C_DIS
LIN {X 109.989,Y 98.688,Z 72.811,A 180.000,B 0.000,C 180.000} C_DIS
LIN {X 110.005,Y 98.532,Z 72.806,A 180.000,B 0.000,C 180.000} C_DIS
LIN {X 110.029,Y 98.298,Z 72.798,A 180.000,B 0.000,C 180.000} C_DIS
LIN {X 110.036,Y 98.222,Z 72.795,A 180.000,B 0.000,C 180.000} C_DIS
LIN {X 110.040,Y 98.145,Z 72.792,A 180.000,B 0.000,C 180.000} C_DIS
LIN {X 110.044,Y 98.068,Z 72.790,A 180.000,B 0.000,C 180.000} C_DIS
LIN {X 110.051,Y 97.911,Z 72.784,A 180.000,B 0.000,C 180.000} C_DIS
LIN {X 110.061,Y 97.676,Z 72.776,A 180.000,B 0.000,C 180.000} C_DIS
LIN {X 110.065,Y 97.598,Z 72.773,A 180.000,B 0.000,C 180.000} C_DIS
LIN {X 110.067,Y 97.520,Z 72.770,A 180.000,B 0.000,C 180.000} C_DIS
LIN {X 110.068,Y 97.442,Z 72.768,A 180.000,B 0.000,C 180.000} C_DIS
LIN {X 110.068,Y 97.364,Z 72.765,A 180.000,B 0.000,C 180.000} C_DIS
LIN {X 110.066,Y 97.209,Z 72.760,A 180.000,B 0.000,C 180.000} C_DIS
LIN {X 110.065,Y 97.131,Z 72.757,A 180.000,B 0.000,C 180.000} C_DIS
LIN {X 110.063,Y 96.975,Z 72.751,A 180.000,B 0.000,C 180.000} C_DIS
LIN {X 110.062,Y 96.896,Z 72.749,A 180.000,B 0.000,C 180.000} C_DIS
LIN {X 110.061,Y 96.818,Z 72.746,A 180.000,B 0.000,C 180.000} C_DIS
LIN {X 110.057,Y 96.741,Z 72.743,A 180.000,B 0.000,C 180.000} C_DIS
LIN {X 110.052,Y 96.663,Z 72.741,A 180.000,B 0.000,C 180.000} C_DIS
LIN {X 110.036,Y 96.429,Z 72.732,A 180.000,B 0.000,C 180.000} C_DIS
LIN {X 110.026,Y 96.273,Z 72.727,A 180.000,B 0.000,C 180.000} C_DIS
LIN {X 110.020,Y 96.194,Z 72.724,A 180.000,B 0.000,C 180.000} C_DIS
LIN {X 110.014,Y 96.117,Z 72.721,A 180.000,B 0.000,C 180.000} C_DIS
LIN {X 110.006,Y 96.040,Z 72.719,A 180.000,B 0.000,C 180.000} C_DIS
LIN {X 109.997,Y 95.963,Z 72.716,A 180.000,B 0.000,C 180.000} C_DIS
LIN {X 109.987,Y 95.886,Z 72.713,A 180.000,B 0.000,C 180.000} C_DIS
LIN {X 109.968,Y 95.730,Z 72.708,A 180.000,B 0.000,C 180.000} C_DIS
LIN {X 109.939,Y 95.497,Z 72.700,A 180.000,B 0.000,C 180.000} C_DIS
LIN {X 109.929,Y 95.420,Z 72.697,A 180.000,B 0.000,C 180.000} C_DIS
LIN {X 109.917,Y 95.343,Z 72.694,A 180.000,B 0.000,C 180.000} C_DIS
LIN {X 109.904,Y 95.267,Z 72.692,A 180.000,B 0.000,C 180.000} C_DIS
LIN {X 109.890,Y 95.189,Z 72.689,A 180.000,B 0.000,C 180.000} C_DIS
LIN {X 109.875,Y 95.112,Z 72.686,A 180.000,B 0.000,C 180.000} C_DIS
LIN {X 109.861,Y 95.034,Z 72.683,A 180.000,B 0.000,C 180.000} C_DIS
LIN {X 109.847,Y 94.957,Z 72.681,A 180.000,B 0.000,C 180.000} C_DIS
LIN {X 109.833,Y 94.880,Z 72.678,A 180.000,B 0.000,C 180.000} C_DIS
LIN {X 109.819,Y 94.803,Z 72.675,A 180.000,B 0.000,C 180.000} C_DIS
LIN {X 109.805,Y 94.727,Z 72.673,A 180.000,B 0.000,C 180.000} C_DIS
LIN {X 109.788,Y 94.651,Z 72.670,A 180.000,B 0.000,C 180.000} C_DIS
LIN {X 109.769,Y 94.574,Z 72.668,A 180.000,B 0.000,C 180.000} C_DIS
LIN {X 109.751,Y 94.498,Z 72.665,A 180.000,B 0.000,C 180.000} C_DIS
LIN {X 109.732,Y 94.422,Z 72.662,A 180.000,B 0.000,C 180.000} C_DIS
LIN {X 109.714,Y 94.346,Z 72.660,A 180.000,B 0.000,C 180.000} C_DIS
LIN {X 109.696,Y 94.270,Z 72.657,A 180.000,B 0.000,C 180.000} C_DIS
LIN {X 109.677,Y 94.194,Z 72.655,A 180.000,B 0.000,C 180.000} C_DIS
LIN {X 109.640,Y 94.042,Z 72.650,A 180.000,B 0.000,C 180.000} C_DIS
LIN {X 109.598,Y 93.891,Z 72.645,A 180.000,B 0.000,C 180.000} C_DIS
LIN {X 109.553,Y 93.741,Z 72.640,A 180.000,B 0.000,C 180.000} C_DIS
LIN {X 109.507,Y 93.590,Z 72.635,A 180.000,B 0.000,C 180.000} C_DIS
LIN {X 109.461,Y 93.440,Z 72.630,A 180.000,B 0.000,C 180.000} C_DIS
LIN {X 109.413,Y 93.291,Z 72.626,A 180.000,B 0.000,C 180.000} C_DIS
LIN {X 109.360,Y 93.145,Z 72.621,A 180.000,B 0.000,C 180.000} C_DIS
LIN {X 109.306,Y 92.997,Z 72.616,A 180.000,B 0.000,C 180.000} C_DIS
LIN {X 109.251,Y 92.849,Z 72.612,A 180.000,B 0.000,C 180.000} C_DIS
LIN {X 109.197,Y 92.703,Z 72.607,A 180.000,B 0.000,C 180.000} C_DIS
LIN {X 109.139,Y 92.558,Z 72.603,A 180.000,B 0.000,C 180.000} C_DIS
LIN {X 109.076,Y 92.413,Z 72.599,A 180.000,B 0.000,C 180.000} C_DIS
LIN {X 109.014,Y 92.269,Z 72.595,A 180.000,B 0.000,C 180.000} C_DIS
LIN {X 108.951,Y 92.125,Z 72.590,A 180.000,B 0.000,C 180.000} C_DIS
LIN {X 108.887,Y 91.982,Z 72.586,A 180.000,B 0.000,C 180.000} C_DIS
LIN {X 108.817,Y 91.841,Z 72.582,A 180.000,B 0.000,C 180.000} C_DIS
LIN {X 108.746,Y 91.701,Z 72.579,A 180.000,B 0.000,C 180.000} C_DIS
LIN {X 108.676,Y 91.560,Z 72.575,A 180.000,B 0.000,C 180.000} C_DIS
LIN {X 108.604,Y 91.420,Z 72.571,A 180.000,B 0.000,C 180.000} C_DIS
LIN {X 108.529,Y 91.282,Z 72.567,A 180.000,B 0.000,C 180.000} C_DIS
LIN {X 108.451,Y 91.147,Z 72.564,A 180.000,B 0.000,C 180.000} C_DIS
LIN {X 108.372,Y 91.010,Z 72.560,A 180.000,B 0.000,C 180.000} C_DIS
LIN {X 108.294,Y 90.874,Z 72.557,A 180.000,B 0.000,C 180.000} C_DIS
LIN {X 108.214,Y 90.739,Z 72.554,A 180.000,B 0.000,C 180.000} C_DIS
LIN {X 108.128,Y 90.607,Z 72.550,A 180.000,B 0.000,C 180.000} C_DIS
LIN {X 108.042,Y 90.475,Z 72.547,A 180.000,B 0.000,C 180.000} C_DIS
LIN {X 107.956,Y 90.344,Z 72.544,A 180.000,B 0.000,C 180.000} C_DIS
LIN {X 107.869,Y 90.213,Z 72.541,A 180.000,B 0.000,C 180.000} C_DIS
LIN {X 107.779,Y 90.084,Z 72.538,A 180.000,B 0.000,C 180.000} C_DIS
LIN {X 107.685,Y 89.958,Z 72.536,A 180.000,B 0.000,C 180.000} C_DIS
LIN {X 107.591,Y 89.831,Z 72.533,A 180.000,B 0.000,C 180.000} C_DIS
LIN {X 107.498,Y 89.705,Z 72.530,A 180.000,B 0.000,C 180.000} C_DIS
LIN {X 107.403,Y 89.579,Z 72.528,A 180.000,B 0.000,C 180.000} C_DIS
LIN {X 107.202,Y 89.337,Z 72.523,A 180.000,B 0.000,C 180.000} C_DIS
LIN {X 107.000,Y 89.095,Z 72.519,A 180.000,B 0.000,C 180.000} C_DIS
LIN {X 106.788,Y 88.863,Z 72.515,A 180.000,B 0.000,C 180.000} C_DIS
LIN {X 106.572,Y 88.633,Z 72.512,A 180.000,B 0.000,C 180.000} C_DIS
LIN {X 106.351,Y 88.410,Z 72.509,A 180.000,B 0.000,C 180.000} C_DIS
LIN {X 106.123,Y 88.192,Z 72.506,A 180.000,B 0.000,C 180.000} C_DIS
LIN {X 105.891,Y 87.980,Z 72.504,A 180.000,B 0.000,C 180.000} C_DIS
LIN {X 105.651,Y 87.776,Z 72.502,A 180.000,B 0.000,C 180.000} C_DIS
LIN {X 105.410,Y 87.573,Z 72.501,A 180.000,B 0.000,C 180.000} C_DIS
LIN {X 105.159,Y 87.382,Z 72.500,A 180.000,B 0.000,C 180.000} C_DIS
LIN {X 104.913,Y 87.198,Z 72.500,A 180.000,B 0.000,C 180.000} C_DIS
; Cutting Move Starts
LIN {X 104.762,Y 87.091,Z 72.500,A 180.000,B 0.000,C 180.000} C_DIS
LIN {X 104.405,Y 86.852,Z 72.500,A 180.000,B 0.000,C 180.000} C_DIS
LIN {X 104.226,Y 86.735,Z 72.500,A 180.000,B 0.000,C 180.000} C_DIS
LIN {X 104.179,Y 86.707,Z 72.500,A 180.000,B 0.000,C 180.000} C_DIS
LIN {X 104.047,Y 86.629,Z 72.500,A 180.000,B 0.000,C 180.000} C_DIS
LIN {X 103.869,Y 86.523,Z 72.500,A 180.000,B 0.000,C 180.000} C_DIS
LIN {X 103.690,Y 86.418,Z 72.500,A 180.000,B 0.000,C 180.000} C_DIS
LIN {X 103.564,Y 86.349,Z 72.500,A 180.000,B 0.000,C 180.000} C_DIS
LIN {X 103.153,Y 86.137,Z 72.500,A 180.000,B 0.000,C 180.000} C_DIS
LIN {X 102.975,Y 86.049,Z 72.500,A 180.000,B 0.000,C 180.000} C_DIS
LIN {X 102.850,Y 85.992,Z 72.500,A 180.000,B 0.000,C 180.000} C_DIS
LIN {X 102.438,Y 85.808,Z 72.500,A 180.000,B 0.000,C 180.000} C_DIS
LIN {X 102.260,Y 85.733,Z 72.500,A 180.000,B 0.000,C 180.000} C_DIS
LIN {X 101.902,Y 85.597,Z 72.500,A 180.000,B 0.000,C 180.000} C_DIS
LIN {X 101.723,Y 85.530,Z 72.500,A 180.000,B 0.000,C 180.000} C_DIS
LIN {X 101.545,Y 85.471,Z 72.500,A 180.000,B 0.000,C 180.000} C_DIS
LIN {X 101.187,Y 85.357,Z 72.500,A 180.000,B 0.000,C 180.000} C_DIS
LIN {X 101.008,Y 85.301,Z 72.500,A 180.000,B 0.000,C 180.000} C_DIS
LIN {X 100.920,Y 85.276,Z 72.500,A 180.000,B 0.000,C 180.000} C_DIS
LIN {X 100.472,Y 85.161,Z 72.500,A 180.000,B 0.000,C 180.000} C_DIS
LIN {X 100.293,Y 85.118,Z 72.500,A 180.000,B 0.000,C 180.000} C_DIS
LIN {X 100.193,Y 85.098,Z 72.500,A 180.000,B 0.000,C 180.000} C_DIS
LIN {X 99.757,Y 85.011,Z 72.500,A 180.000,B 0.000,C 180.000} C_DIS
LIN {X 99.578,Y 84.978,Z 72.500,A 180.000,B 0.000,C 180.000} C_DIS
LIN {X 99.399,Y 84.952,Z 72.500,A 180.000,B 0.000,C 180.000} C_DIS
LIN {X 99.042,Y 84.902,Z 72.500,A 180.000,B 0.000,C 180.000} C_DIS
LIN {X 98.863,Y 84.880,Z 72.500,A 180.000,B 0.000,C 180.000} C_DIS
LIN {X 98.327,Y 84.835,Z 72.500,A 180.000,B 0.000,C 180.000} C_DIS
LIN {X 98.148,Y 84.823,Z 72.500,A 180.000,B 0.000,C 180.000} C_DIS
LIN {X 97.969,Y 84.818,Z 72.500,A 180.000,B 0.000,C 180.000} C_DIS
LIN {X 97.612,Y 84.808,Z 72.500,A 180.000,B 0.000,C 180.000} C_DIS
LIN {X 97.433,Y 84.807,Z 72.500,A 180.000,B 0.000,C 180.000} C_DIS
LIN {X 96.897,Y 84.822,Z 72.500,A 180.000,B 0.000,C 180.000} C_DIS
LIN {X 96.718,Y 84.831,Z 72.500,A 180.000,B 0.000,C 180.000} C_DIS
LIN {X 96.539,Y 84.846,Z 72.500,A 180.000,B 0.000,C 180.000} C_DIS
LIN {X 96.181,Y 84.876,Z 72.500,A 180.000,B 0.000,C 180.000} C_DIS
LIN {X 96.003,Y 84.895,Z 72.500,A 180.000,B 0.000,C 180.000} C_DIS
LIN {X 95.466,Y 84.971,Z 72.500,A 180.000,B 0.000,C 180.000} C_DIS
LIN {X 95.288,Y 85.002,Z 72.500,A 180.000,B 0.000,C 180.000} C_DIS
LIN {X 95.109,Y 85.038,Z 72.500,A 180.000,B 0.000,C 180.000} C_DIS
LIN {X 94.751,Y 85.109,Z 72.500,A 180.000,B 0.000,C 180.000} C_DIS
LIN {X 94.573,Y 85.149,Z 72.500,A 180.000,B 0.000,C 180.000} C_DIS
LIN {X 94.080,Y 85.276,Z 72.500,A 180.000,B 0.000,C 180.000} C_DIS
LIN {X 94.036,Y 85.288,Z 72.500,A 180.000,B 0.000,C 180.000} C_DIS
LIN {X 93.857,Y 85.343,Z 72.500,A 180.000,B 0.000,C 180.000} C_DIS
LIN {X 93.500,Y 85.457,Z 72.500,A 180.000,B 0.000,C 180.000} C_DIS
LIN {X 93.321,Y 85.514,Z 72.500,A 180.000,B 0.000,C 180.000} C_DIS
LIN {X 93.142,Y 85.580,Z 72.500,A 180.000,B 0.000,C 180.000} C_DIS
LIN {X 92.785,Y 85.717,Z 72.500,A 180.000,B 0.000,C 180.000} C_DIS
LIN {X 92.606,Y 85.788,Z 72.500,A 180.000,B 0.000,C 180.000} C_DIS
LIN {X 92.550,Y 85.813,Z 72.500,A 180.000,B 0.000,C 180.000} C_DIS
LIN {X 92.150,Y 85.992,Z 72.500,A 180.000,B 0.000,C 180.000} C_DIS
LIN {X 92.070,Y 86.028,Z 72.500,A 180.000,B 0.000,C 180.000} C_DIS
LIN {X 91.891,Y 86.114,Z 72.500,A 180.000,B 0.000,C 180.000} C_DIS
LIN {X 91.436,Y 86.349,Z 72.500,A 180.000,B 0.000,C 180.000} C_DIS
LIN {X 91.355,Y 86.393,Z 72.500,A 180.000,B 0.000,C 180.000} C_DIS
LIN {X 91.176,Y 86.497,Z 72.500,A 180.000,B 0.000,C 180.000} C_DIS
LIN {X 90.997,Y 86.603,Z 72.500,A 180.000,B 0.000,C 180.000} C_DIS
LIN {X 90.821,Y 86.707,Z 72.500,A 180.000,B 0.000,C 180.000} C_DIS
LIN {X 90.818,Y 86.708,Z 72.500,A 180.000,B 0.000,C 180.000} C_DIS
LIN {X 90.640,Y 86.822,Z 72.500,A 180.000,B 0.000,C 180.000} C_DIS
LIN {X 90.277,Y 87.064,Z 72.500,A 180.000,B 0.000,C 180.000} C_DIS
LIN {X 90.103,Y 87.184,Z 72.500,A 180.000,B 0.000,C 180.000} C_DIS
LIN {X 90.025,Y 87.243,Z 72.500,A 180.000,B 0.000,C 180.000} C_DIS
LIN {X 89.746,Y 87.453,Z 72.500,A 180.000,B 0.000,C 180.000} C_DIS
LIN {X 89.567,Y 87.591,Z 72.500,A 180.000,B 0.000,C 180.000} C_DIS
LIN {X 89.556,Y 87.601,Z 72.500,A 180.000,B 0.000,C 180.000} C_DIS
LIN {X 89.388,Y 87.741,Z 72.500,A 180.000,B 0.000,C 180.000} C_DIS
LIN {X 89.132,Y 87.958,Z 72.500,A 180.000,B 0.000,C 180.000} C_DIS
LIN {X 89.031,Y 88.045,Z 72.500,A 180.000,B 0.000,C 180.000} C_DIS
LIN {X 88.932,Y 88.137,Z 72.500,A 180.000,B 0.000,C 180.000} C_DIS
LIN {X 88.673,Y 88.381,Z 72.500,A 180.000,B 0.000,C 180.000} C_DIS
LIN {X 88.554,Y 88.494,Z 72.500,A 180.000,B 0.000,C 180.000} C_DIS
LIN {X 88.494,Y 88.555,Z 72.500,A 180.000,B 0.000,C 180.000} C_DIS
LIN {X 88.383,Y 88.673,Z 72.500,A 180.000,B 0.000,C 180.000} C_DIS
LIN {X 88.137,Y 88.933,Z 72.500,A 180.000,B 0.000,C 180.000} C_DIS
LIN {X 88.045,Y 89.031,Z 72.500,A 180.000,B 0.000,C 180.000} C_DIS
LIN {X 87.958,Y 89.130,Z 72.500,A 180.000,B 0.000,C 180.000} C_DIS
LIN {X 87.740,Y 89.388,Z 72.500,A 180.000,B 0.000,C 180.000} C_DIS
LIN {X 87.601,Y 89.554,Z 72.500,A 180.000,B 0.000,C 180.000} C_DIS
LIN {X 87.590,Y 89.567,Z 72.500,A 180.000,B 0.000,C 180.000} C_DIS
LIN {X 87.454,Y 89.746,Z 72.500,A 180.000,B 0.000,C 180.000} C_DIS
LIN {X 87.243,Y 90.026,Z 72.500,A 180.000,B 0.000,C 180.000} C_DIS
LIN {X 87.185,Y 90.103,Z 72.500,A 180.000,B 0.000,C 180.000} C_DIS
LIN {X 87.064,Y 90.277,Z 72.500,A 180.000,B 0.000,C 180.000} C_DIS
LIN {X 86.822,Y 90.640,Z 72.500,A 180.000,B 0.000,C 180.000} C_DIS
LIN {X 86.708,Y 90.818,Z 72.500,A 180.000,B 0.000,C 180.000} C_DIS
LIN {X 86.497,Y 91.176,Z 72.500,A 180.000,B 0.000,C 180.000} C_DIS
LIN {X 86.394,Y 91.355,Z 72.500,A 180.000,B 0.000,C 180.000} C_DIS
LIN {X 86.349,Y 91.437,Z 72.500,A 180.000,B 0.000,C 180.000} C_DIS
LIN {X 86.299,Y 91.533,Z 72.500,A 180.000,B 0.000,C 180.000} C_DIS
LIN {X 86.114,Y 91.891,Z 72.500,A 180.000,B 0.000,C 180.000} C_DIS
LIN {X 86.027,Y 92.070,Z 72.500,A 180.000,B 0.000,C 180.000} C_DIS
LIN {X 85.813,Y 92.549,Z 72.500,A 180.000,B 0.000,C 180.000} C_DIS
LIN {X 85.788,Y 92.606,Z 72.500,A 180.000,B 0.000,C 180.000} C_DIS
LIN {X 85.717,Y 92.785,Z 72.500,A 180.000,B 0.000,C 180.000} C_DIS
LIN {X 85.581,Y 93.142,Z 72.500,A 180.000,B 0.000,C 180.000} C_DIS
LIN {X 85.514,Y 93.321,Z 72.500,A 180.000,B 0.000,C 180.000} C_DIS
LIN {X 85.456,Y 93.500,Z 72.500,A 180.000,B 0.000,C 180.000} C_DIS
LIN {X 85.342,Y 93.857,Z 72.500,A 180.000,B 0.000,C 180.000} C_DIS
LIN {X 85.289,Y 94.036,Z 72.500,A 180.000,B 0.000,C 180.000} C_DIS
LIN {X 85.197,Y 94.394,Z 72.500,A 180.000,B 0.000,C 180.000} C_DIS
LIN {X 85.151,Y 94.573,Z 72.500,A 180.000,B 0.000,C 180.000} C_DIS
LIN {X 85.108,Y 94.751,Z 72.500,A 180.000,B 0.000,C 180.000} C_DIS
LIN {X 85.098,Y 94.802,Z 72.500,A 180.000,B 0.000,C 180.000} C_DIS
LIN {X 85.001,Y 95.288,Z 72.500,A 180.000,B 0.000,C 180.000} C_DIS
LIN {X 84.972,Y 95.466,Z 72.500,A 180.000,B 0.000,C 180.000} C_DIS
LIN {X 84.919,Y 95.840,Z 72.500,A 180.000,B 0.000,C 180.000} C_DIS
LIN {X 84.896,Y 96.003,Z 72.500,A 180.000,B 0.000,C 180.000} C_DIS
LIN {X 84.876,Y 96.181,Z 72.500,A 180.000,B 0.000,C 180.000} C_DIS
LIN {X 84.831,Y 96.718,Z 72.500,A 180.000,B 0.000,C 180.000} C_DIS
LIN {X 84.822,Y 96.897,Z 72.500,A 180.000,B 0.000,C 180.000} C_DIS
LIN {X 84.812,Y 97.254,Z 72.500,A 180.000,B 0.000,C 180.000} C_DIS
LIN {X 84.807,Y 97.433,Z 72.500,A 180.000,B 0.000,C 180.000} C_DIS
LIN {X 84.808,Y 97.612,Z 72.500,A 180.000,B 0.000,C 180.000} C_DIS
LIN {X 84.823,Y 98.148,Z 72.500,A 180.000,B 0.000,C 180.000} C_DIS
LIN {X 84.835,Y 98.327,Z 72.500,A 180.000,B 0.000,C 180.000} C_DIS
LIN {X 84.865,Y 98.684,Z 72.500,A 180.000,B 0.000,C 180.000} C_DIS
LIN {X 84.880,Y 98.863,Z 72.500,A 180.000,B 0.000,C 180.000} C_DIS
LIN {X 84.902,Y 99.042,Z 72.500,A 180.000,B 0.000,C 180.000} C_DIS
LIN {X 84.953,Y 99.399,Z 72.500,A 180.000,B 0.000,C 180.000} C_DIS
LIN {X 84.978,Y 99.578,Z 72.500,A 180.000,B 0.000,C 180.000} C_DIS
LIN {X 85.010,Y 99.757,Z 72.500,A 180.000,B 0.000,C 180.000} C_DIS
LIN {X 85.098,Y 100.198,Z 72.500,A 180.000,B 0.000,C 180.000} C_DIS
LIN {X 85.117,Y 100.293,Z 72.500,A 180.000,B 0.000,C 180.000} C_DIS
LIN {X 85.162,Y 100.472,Z 72.500,A 180.000,B 0.000,C 180.000} C_DIS
LIN {X 85.276,Y 100.916,Z 72.500,A 180.000,B 0.000,C 180.000} C_DIS
LIN {X 85.301,Y 101.008,Z 72.500,A 180.000,B 0.000,C 180.000} C_DIS
LIN {X 85.356,Y 101.187,Z 72.500,A 180.000,B 0.000,C 180.000} C_DIS
LIN {X 85.470,Y 101.545,Z 72.500,A 180.000,B 0.000,C 180.000} C_DIS
LIN {X 85.530,Y 101.723,Z 72.500,A 180.000,B 0.000,C 180.000} C_DIS
LIN {X 85.598,Y 101.902,Z 72.500,A 180.000,B 0.000,C 180.000} C_DIS
LIN {X 85.666,Y 102.081,Z 72.500,A 180.000,B 0.000,C 180.000} C_DIS
LIN {X 85.734,Y 102.260,Z 72.500,A 180.000,B 0.000,C 180.000} C_DIS
LIN {X 85.807,Y 102.438,Z 72.500,A 180.000,B 0.000,C 180.000} C_DIS
LIN {X 85.813,Y 102.451,Z 72.500,A 180.000,B 0.000,C 180.000} C_DIS
LIN {X 85.992,Y 102.851,Z 72.500,A 180.000,B 0.000,C 180.000} C_DIS
LIN {X 86.047,Y 102.975,Z 72.500,A 180.000,B 0.000,C 180.000} C_DIS
LIN {X 86.137,Y 103.153,Z 72.500,A 180.000,B 0.000,C 180.000} C_DIS
LIN {X 86.322,Y 103.511,Z 72.500,A 180.000,B 0.000,C 180.000} C_DIS
LIN {X 86.349,Y 103.563,Z 72.500,A 180.000,B 0.000,C 180.000} C_DIS
LIN {X 86.418,Y 103.690,Z 72.500,A 180.000,B 0.000,C 180.000} C_DIS
LIN {X 86.523,Y 103.869,Z 72.500,A 180.000,B 0.000,C 180.000} C_DIS
LIN {X 86.707,Y 104.179,Z 72.500,A 180.000,B 0.000,C 180.000} C_DIS
LIN {X 86.735,Y 104.226,Z 72.500,A 180.000,B 0.000,C 180.000} C_DIS
LIN {X 86.851,Y 104.405,Z 72.500,A 180.000,B 0.000,C 180.000} C_DIS
LIN {X 87.090,Y 104.762,Z 72.500,A 180.000,B 0.000,C 180.000} C_DIS
LIN {X 87.218,Y 104.941,Z 72.500,A 180.000,B 0.000,C 180.000} C_DIS
LIN {X 87.487,Y 105.299,Z 72.500,A 180.000,B 0.000,C 180.000} C_DIS
LIN {X 87.601,Y 105.446,Z 72.500,A 180.000,B 0.000,C 180.000} C_DIS
LIN {X 87.627,Y 105.477,Z 72.500,A 180.000,B 0.000,C 180.000} C_DIS
LIN {X 87.958,Y 105.870,Z 72.500,A 180.000,B 0.000,C 180.000} C_DIS
LIN {X 88.087,Y 106.014,Z 72.500,A 180.000,B 0.000,C 180.000} C_DIS
LIN {X 88.137,Y 106.067,Z 72.500,A 180.000,B 0.000,C 180.000} C_DIS
LIN {X 88.425,Y 106.371,Z 72.500,A 180.000,B 0.000,C 180.000} C_DIS
LIN {X 88.494,Y 106.445,Z 72.500,A 180.000,B 0.000,C 180.000} C_DIS
LIN {X 88.600,Y 106.550,Z 72.500,A 180.000,B 0.000,C 180.000} C_DIS
LIN {X 88.979,Y 106.908,Z 72.500,A 180.000,B 0.000,C 180.000} C_DIS
LIN {X 89.031,Y 106.955,Z 72.500,A 180.000,B 0.000,C 180.000} C_DIS
LIN {X 89.184,Y 107.086,Z 72.500,A 180.000,B 0.000,C 180.000} C_DIS
LIN {X 89.396,Y 107.265,Z 72.500,A 180.000,B 0.000,C 180.000} C_DIS
LIN {X 89.567,Y 107.409,Z 72.500,A 180.000,B 0.000,C 180.000} C_DIS
LIN {X 89.611,Y 107.444,Z 72.500,A 180.000,B 0.000,C 180.000} C_DIS
LIN {X 89.746,Y 107.547,Z 72.500,A 180.000,B 0.000,C 180.000} C_DIS
LIN {X 90.084,Y 107.802,Z 72.500,A 180.000,B 0.000,C 180.000} C_DIS
LIN {X 90.103,Y 107.816,Z 72.500,A 180.000,B 0.000,C 180.000} C_DIS
LIN {X 90.282,Y 107.939,Z 72.500,A 180.000,B 0.000,C 180.000} C_DIS
LIN {X 90.640,Y 108.178,Z 72.500,A 180.000,B 0.000,C 180.000} C_DIS
LIN {X 90.818,Y 108.292,Z 72.500,A 180.000,B 0.000,C 180.000} C_DIS
LIN {X 90.896,Y 108.338,Z 72.500,A 180.000,B 0.000,C 180.000} C_DIS
LIN {X 91.199,Y 108.517,Z 72.500,A 180.000,B 0.000,C 180.000} C_DIS
LIN {X 91.355,Y 108.607,Z 72.500,A 180.000,B 0.000,C 180.000} C_DIS
LIN {X 91.522,Y 108.695,Z 72.500,A 180.000,B 0.000,C 180.000} C_DIS
LIN {X 91.868,Y 108.874,Z 72.500,A 180.000,B 0.000,C 180.000} C_DIS
LIN {X 91.891,Y 108.886,Z 72.500,A 180.000,B 0.000,C 180.000} C_DIS
LIN {X 92.070,Y 108.972,Z 72.500,A 180.000,B 0.000,C 180.000} C_DIS
LIN {X 92.250,Y 109.053,Z 72.500,A 180.000,B 0.000,C 180.000} C_DIS
LIN {X 92.427,Y 109.132,Z 72.500,A 180.000,B 0.000,C 180.000} C_DIS
LIN {X 92.606,Y 109.212,Z 72.500,A 180.000,B 0.000,C 180.000} C_DIS
LIN {X 92.652,Y 109.232,Z 72.500,A 180.000,B 0.000,C 180.000} C_DIS
LIN {X 92.785,Y 109.283,Z 72.500,A 180.000,B 0.000,C 180.000} C_DIS
LIN {X 93.142,Y 109.420,Z 72.500,A 180.000,B 0.000,C 180.000} C_DIS
LIN {X 93.321,Y 109.486,Z 72.500,A 180.000,B 0.000,C 180.000} C_DIS
LIN {X 93.500,Y 109.543,Z 72.500,A 180.000,B 0.000,C 180.000} C_DIS
LIN {X 93.857,Y 109.657,Z 72.500,A 180.000,B 0.000,C 180.000} C_DIS
LIN {X 94.036,Y 109.712,Z 72.500,A 180.000,B 0.000,C 180.000} C_DIS
LIN {X 94.215,Y 109.758,Z 72.500,A 180.000,B 0.000,C 180.000} C_DIS
LIN {X 94.573,Y 109.851,Z 72.500,A 180.000,B 0.000,C 180.000} C_DIS
LIN {X 94.751,Y 109.891,Z 72.500,A 180.000,B 0.000,C 180.000} C_DIS
LIN {X 95.109,Y 109.962,Z 72.500,A 180.000,B 0.000,C 180.000} C_DIS
LIN {X 95.288,Y 109.998,Z 72.500,A 180.000,B 0.000,C 180.000} C_DIS
LIN {X 95.466,Y 110.029,Z 72.500,A 180.000,B 0.000,C 180.000} C_DIS
LIN {X 96.003,Y 110.105,Z 72.500,A 180.000,B 0.000,C 180.000} C_DIS
LIN {X 96.181,Y 110.124,Z 72.500,A 180.000,B 0.000,C 180.000} C_DIS
LIN {X 96.539,Y 110.154,Z 72.500,A 180.000,B 0.000,C 180.000} C_DIS
LIN {X 96.718,Y 110.169,Z 72.500,A 180.000,B 0.000,C 180.000} C_DIS
LIN {X 96.897,Y 110.178,Z 72.500,A 180.000,B 0.000,C 180.000} C_DIS
LIN {X 97.433,Y 110.193,Z 72.500,A 180.000,B 0.000,C 180.000} C_DIS
LIN {X 97.612,Y 110.192,Z 72.500,A 180.000,B 0.000,C 180.000} C_DIS
LIN {X 97.969,Y 110.182,Z 72.500,A 180.000,B 0.000,C 180.000} C_DIS
LIN {X 98.148,Y 110.177,Z 72.500,A 180.000,B 0.000,C 180.000} C_DIS
LIN {X 98.327,Y 110.165,Z 72.500,A 180.000,B 0.000,C 180.000} C_DIS
LIN {X 98.863,Y 110.120,Z 72.500,A 180.000,B 0.000,C 180.000} C_DIS
LIN {X 99.042,Y 110.098,Z 72.500,A 180.000,B 0.000,C 180.000} C_DIS
LIN {X 99.399,Y 110.048,Z 72.500,A 180.000,B 0.000,C 180.000} C_DIS
LIN {X 99.578,Y 110.022,Z 72.500,A 180.000,B 0.000,C 180.000} C_DIS
LIN {X 99.757,Y 109.989,Z 72.500,A 180.000,B 0.000,C 180.000} C_DIS
LIN {X 100.114,Y 109.918,Z 72.500,A 180.000,B 0.000,C 180.000} C_DIS
LIN {X 100.293,Y 109.882,Z 72.500,A 180.000,B 0.000,C 180.000} C_DIS
LIN {X 100.472,Y 109.839,Z 72.500,A 180.000,B 0.000,C 180.000} C_DIS
LIN {X 100.829,Y 109.747,Z 72.500,A 180.000,B 0.000,C 180.000} C_DIS
LIN {X 101.008,Y 109.699,Z 72.500,A 180.000,B 0.000,C 180.000} C_DIS
LIN {X 101.187,Y 109.643,Z 72.500,A 180.000,B 0.000,C 180.000} C_DIS
LIN {X 101.545,Y 109.529,Z 72.500,A 180.000,B 0.000,C 180.000} C_DIS
LIN {X 101.723,Y 109.470,Z 72.500,A 180.000,B 0.000,C 180.000} C_DIS
LIN {X 101.883,Y 109.410,Z 72.500,A 180.000,B 0.000,C 180.000} C_DIS
LIN {X 102.260,Y 109.267,Z 72.500,A 180.000,B 0.000,C 180.000} C_DIS
LIN {X 102.348,Y 109.232,Z 72.500,A 180.000,B 0.000,C 180.000} C_DIS
LIN {X 102.438,Y 109.192,Z 72.500,A 180.000,B 0.000,C 180.000} C_DIS
LIN {X 102.796,Y 109.032,Z 72.500,A 180.000,B 0.000,C 180.000} C_DIS
LIN {X 102.975,Y 108.951,Z 72.500,A 180.000,B 0.000,C 180.000} C_DIS
LIN {X 103.132,Y 108.874,Z 72.500,A 180.000,B 0.000,C 180.000} C_DIS
LIN {X 103.511,Y 108.678,Z 72.500,A 180.000,B 0.000,C 180.000} C_DIS
LIN {X 103.690,Y 108.582,Z 72.500,A 180.000,B 0.000,C 180.000} C_DIS
LIN {X 103.801,Y 108.517,Z 72.500,A 180.000,B 0.000,C 180.000} C_DIS
LIN {X 104.104,Y 108.338,Z 72.500,A 180.000,B 0.000,C 180.000} C_DIS
LIN {X 104.226,Y 108.265,Z 72.500,A 180.000,B 0.000,C 180.000} C_DIS
LIN {X 104.389,Y 108.159,Z 72.500,A 180.000,B 0.000,C 180.000} C_DIS
LIN {X 104.762,Y 107.909,Z 72.500,A 180.000,B 0.000,C 180.000} C_DIS
LIN {X 104.916,Y 107.802,Z 72.500,A 180.000,B 0.000,C 180.000} C_DIS
LIN {X 105.299,Y 107.513,Z 72.500,A 180.000,B 0.000,C 180.000} C_DIS
LIN {X 105.389,Y 107.444,Z 72.500,A 180.000,B 0.000,C 180.000} C_DIS
LIN {X 105.477,Y 107.372,Z 72.500,A 180.000,B 0.000,C 180.000} C_DIS
LIN {X 105.604,Y 107.265,Z 72.500,A 180.000,B 0.000,C 180.000} C_DIS
LIN {X 105.835,Y 107.070,Z 72.500,A 180.000,B 0.000,C 180.000} C_DIS
LIN {X 106.014,Y 106.915,Z 72.500,A 180.000,B 0.000,C 180.000} C_DIS
LIN {X 106.021,Y 106.908,Z 72.500,A 180.000,B 0.000,C 180.000} C_DIS
LIN {X 106.400,Y 106.550,Z 72.500,A 180.000,B 0.000,C 180.000} C_DIS
LIN {X 106.550,Y 106.398,Z 72.500,A 180.000,B 0.000,C 180.000} C_DIS
LIN {X 106.744,Y 106.193,Z 72.500,A 180.000,B 0.000,C 180.000} C_DIS
LIN {X 106.908,Y 106.020,Z 72.500,A 180.000,B 0.000,C 180.000} C_DIS
LIN {X 106.913,Y 106.014,Z 72.500,A 180.000,B 0.000,C 180.000} C_DIS
LIN {X 107.071,Y 105.835,Z 72.500,A 180.000,B 0.000,C 180.000} C_DIS
LIN {X 107.373,Y 105.477,Z 72.500,A 180.000,B 0.000,C 180.000} C_DIS
LIN {X 107.444,Y 105.390,Z 72.500,A 180.000,B 0.000,C 180.000} C_DIS
LIN {X 107.513,Y 105.299,Z 72.500,A 180.000,B 0.000,C 180.000} C_DIS
LIN {X 107.782,Y 104.941,Z 72.500,A 180.000,B 0.000,C 180.000} C_DIS
LIN {X 107.802,Y 104.915,Z 72.500,A 180.000,B 0.000,C 180.000} C_DIS
LIN {X 107.910,Y 104.762,Z 72.500,A 180.000,B 0.000,C 180.000} C_DIS
LIN {X 108.159,Y 104.389,Z 72.500,A 180.000,B 0.000,C 180.000} C_DIS
LIN {X 108.265,Y 104.226,Z 72.500,A 180.000,B 0.000,C 180.000} C_DIS
LIN {X 108.338,Y 104.104,Z 72.500,A 180.000,B 0.000,C 180.000} C_DIS
LIN {X 108.517,Y 103.801,Z 72.500,A 180.000,B 0.000,C 180.000} C_DIS
LIN {X 108.582,Y 103.690,Z 72.500,A 180.000,B 0.000,C 180.000} C_DIS
LIN {X 108.678,Y 103.511,Z 72.500,A 180.000,B 0.000,C 180.000} C_DIS
LIN {X 108.874,Y 103.131,Z 72.500,A 180.000,B 0.000,C 180.000} C_DIS
LIN {X 108.953,Y 102.975,Z 72.500,A 180.000,B 0.000,C 180.000} C_DIS
LIN {X 109.033,Y 102.796,Z 72.500,A 180.000,B 0.000,C 180.000} C_DIS
LIN {X 109.113,Y 102.617,Z 72.500,A 180.000,B 0.000,C 180.000} C_DIS
LIN {X 109.193,Y 102.438,Z 72.500,A 180.000,B 0.000,C 180.000} C_DIS
LIN {X 109.232,Y 102.346,Z 72.500,A 180.000,B 0.000,C 180.000} C_DIS
LIN {X 109.266,Y 102.260,Z 72.500,A 180.000,B 0.000,C 180.000} C_DIS
LIN {X 109.334,Y 102.081,Z 72.500,A 180.000,B 0.000,C 180.000} C_DIS
LIN {X 109.410,Y 101.881,Z 72.500,A 180.000,B 0.000,C 180.000} C_DIS
LIN {X 109.470,Y 101.723,Z 72.500,A 180.000,B 0.000,C 180.000} C_DIS
LIN {X 109.530,Y 101.545,Z 72.500,A 180.000,B 0.000,C 180.000} C_DIS
LIN {X 109.644,Y 101.187,Z 72.500,A 180.000,B 0.000,C 180.000} C_DIS
LIN {X 109.699,Y 101.008,Z 72.500,A 180.000,B 0.000,C 180.000} C_DIS
LIN {X 109.746,Y 100.829,Z 72.500,A 180.000,B 0.000,C 180.000} C_DIS
LIN {X 109.838,Y 100.472,Z 72.500,A 180.000,B 0.000,C 180.000} C_DIS
LIN {X 109.883,Y 100.293,Z 72.500,A 180.000,B 0.000,C 180.000} C_DIS
LIN {X 109.919,Y 100.114,Z 72.500,A 180.000,B 0.000,C 180.000} C_DIS
LIN {X 109.990,Y 99.757,Z 72.500,A 180.000,B 0.000,C 180.000} C_DIS
LIN {X 110.022,Y 99.578,Z 72.500,A 180.000,B 0.000,C 180.000} C_DIS
LIN {X 110.047,Y 99.399,Z 72.500,A 180.000,B 0.000,C 180.000} C_DIS
LIN {X 110.098,Y 99.042,Z 72.500,A 180.000,B 0.000,C 180.000} C_DIS
LIN {X 110.120,Y 98.863,Z 72.500,A 180.000,B 0.000,C 180.000} C_DIS
LIN {X 110.126,Y 98.801,Z 72.500,A 180.000,B 0.000,C 180.000} C_DIS
LIN {X 110.165,Y 98.327,Z 72.500,A 180.000,B 0.000,C 180.000} C_DIS
LIN {X 110.177,Y 98.148,Z 72.500,A 180.000,B 0.000,C 180.000} C_DIS
LIN {X 110.192,Y 97.612,Z 72.500,A 180.000,B 0.000,C 180.000} C_DIS
LIN {X 110.193,Y 97.433,Z 72.500,A 180.000,B 0.000,C 180.000} C_DIS
LIN {X 110.188,Y 97.254,Z 72.500,A 180.000,B 0.000,C 180.000} C_DIS
LIN {X 110.178,Y 96.897,Z 72.500,A 180.000,B 0.000,C 180.000} C_DIS
LIN {X 110.169,Y 96.718,Z 72.500,A 180.000,B 0.000,C 180.000} C_DIS
LIN {X 110.124,Y 96.181,Z 72.500,A 180.000,B 0.000,C 180.000} C_DIS
LIN {X 110.104,Y 96.003,Z 72.500,A 180.000,B 0.000,C 180.000} C_DIS
LIN {X 110.079,Y 95.824,Z 72.500,A 180.000,B 0.000,C 180.000} C_DIS
LIN {X 110.028,Y 95.466,Z 72.500,A 180.000,B 0.000,C 180.000} C_DIS
LIN {X 109.999,Y 95.288,Z 72.500,A 180.000,B 0.000,C 180.000} C_DIS
LIN {X 109.928,Y 94.930,Z 72.500,A 180.000,B 0.000,C 180.000} C_DIS
LIN {X 109.892,Y 94.751,Z 72.500,A 180.000,B 0.000,C 180.000} C_DIS
LIN {X 109.849,Y 94.573,Z 72.500,A 180.000,B 0.000,C 180.000} C_DIS
LIN {X 109.803,Y 94.394,Z 72.500,A 180.000,B 0.000,C 180.000} C_DIS
LIN {X 109.711,Y 94.036,Z 72.500,A 180.000,B 0.000,C 180.000} C_DIS
LIN {X 109.658,Y 93.857,Z 72.500,A 180.000,B 0.000,C 180.000} C_DIS
LIN {X 109.544,Y 93.500,Z 72.500,A 180.000,B 0.000,C 180.000} C_DIS
LIN {X 109.486,Y 93.321,Z 72.500,A 180.000,B 0.000,C 180.000} C_DIS
LIN {X 109.419,Y 93.142,Z 72.500,A 180.000,B 0.000,C 180.000} C_DIS
LIN {X 109.283,Y 92.785,Z 72.500,A 180.000,B 0.000,C 180.000} C_DIS
LIN {X 109.232,Y 92.654,Z 72.500,A 180.000,B 0.000,C 180.000} C_DIS
LIN {X 109.212,Y 92.606,Z 72.500,A 180.000,B 0.000,C 180.000} C_DIS
LIN {X 109.133,Y 92.427,Z 72.500,A 180.000,B 0.000,C 180.000} C_DIS
LIN {X 108.973,Y 92.070,Z 72.500,A 180.000,B 0.000,C 180.000} C_DIS
LIN {X 108.886,Y 91.891,Z 72.500,A 180.000,B 0.000,C 180.000} C_DIS
LIN {X 108.695,Y 91.523,Z 72.500,A 180.000,B 0.000,C 180.000} C_DIS
LIN {X 108.606,Y 91.355,Z 72.500,A 180.000,B 0.000,C 180.000} C_DIS
LIN {X 108.517,Y 91.199,Z 72.500,A 180.000,B 0.000,C 180.000} C_DIS
LIN {X 108.292,Y 90.818,Z 72.500,A 180.000,B 0.000,C 180.000} C_DIS
LIN {X 108.178,Y 90.640,Z 72.500,A 180.000,B 0.000,C 180.000} C_DIS
LIN {X 107.939,Y 90.282,Z 72.500,A 180.000,B 0.000,C 180.000} C_DIS
LIN {X 107.815,Y 90.103,Z 72.500,A 180.000,B 0.000,C 180.000} C_DIS
LIN {X 107.802,Y 90.085,Z 72.500,A 180.000,B 0.000,C 180.000} C_DIS
LIN {X 107.681,Y 89.925,Z 72.500,A 180.000,B 0.000,C 180.000} C_DIS
LIN {X 107.546,Y 89.746,Z 72.500,A 180.000,B 0.000,C 180.000} C_DIS
LIN {X 107.444,Y 89.610,Z 72.500,A 180.000,B 0.000,C 180.000} C_DIS
LIN {X 107.410,Y 89.567,Z 72.500,A 180.000,B 0.000,C 180.000} C_DIS
LIN {X 107.265,Y 89.395,Z 72.500,A 180.000,B 0.000,C 180.000} C_DIS
LIN {X 107.086,Y 89.183,Z 72.500,A 180.000,B 0.000,C 180.000} C_DIS
LIN {X 106.955,Y 89.031,Z 72.500,A 180.000,B 0.000,C 180.000} C_DIS
LIN {X 106.908,Y 88.980,Z 72.500,A 180.000,B 0.000,C 180.000} C_DIS
LIN {X 106.786,Y 88.852,Z 72.500,A 180.000,B 0.000,C 180.000} C_DIS
LIN {X 106.550,Y 88.602,Z 72.500,A 180.000,B 0.000,C 180.000} C_DIS
LIN {X 106.446,Y 88.494,Z 72.500,A 180.000,B 0.000,C 180.000} C_DIS
LIN {X 106.371,Y 88.423,Z 72.500,A 180.000,B 0.000,C 180.000} C_DIS
LIN {X 106.068,Y 88.137,Z 72.500,A 180.000,B 0.000,C 180.000} C_DIS
LIN {X 106.014,Y 88.085,Z 72.500,A 180.000,B 0.000,C 180.000} C_DIS
LIN {X 105.868,Y 87.958,Z 72.500,A 180.000,B 0.000,C 180.000} C_DIS
LIN {X 105.656,Y 87.779,Z 72.500,A 180.000,B 0.000,C 180.000} C_DIS
LIN {X 105.477,Y 87.628,Z 72.500,A 180.000,B 0.000,C 180.000} C_DIS
LIN {X 105.444,Y 87.601,Z 72.500,A 180.000,B 0.000,C 180.000} C_DIS
LIN {X 105.299,Y 87.487,Z 72.500,A 180.000,B 0.000,C 180.000} C_DIS
LIN {X 104.941,Y 87.218,Z 72.500,A 180.000,B 0.000,C 180.000} C_DIS
LIN {X 104.913,Y 87.198,Z 72.500,A 180.000,B 0.000,C 180.000} C_DIS
; Link Move Starts
LIN {X 104.674,Y 87.032,Z 72.500,A 180.000,B 0.000,C 180.000} C_DIS
LIN {X 104.412,Y 86.856,Z 72.499,A 180.000,B 0.000,C 180.000} C_DIS
LIN {X 104.166,Y 86.698,Z 72.498,A 180.000,B 0.000,C 180.000} C_DIS
LIN {X 103.899,Y 86.539,Z 72.496,A 180.000,B 0.000,C 180.000} C_DIS
LIN {X 103.648,Y 86.391,Z 72.495,A 180.000,B 0.000,C 180.000} C_DIS
LIN {X 103.371,Y 86.245,Z 72.492,A 180.000,B 0.000,C 180.000} C_DIS
LIN {X 103.099,Y 86.103,Z 72.489,A 180.000,B 0.000,C 180.000} C_DIS
LIN {X 102.830,Y 85.976,Z 72.486,A 180.000,B 0.000,C 180.000} C_DIS
LIN {X 102.544,Y 85.846,Z 72.482,A 180.000,B 0.000,C 180.000} C_DIS
LIN {X 102.270,Y 85.727,Z 72.478,A 180.000,B 0.000,C 180.000} C_DIS
LIN {X 101.985,Y 85.616,Z 72.474,A 180.000,B 0.000,C 180.000} C_DIS
LIN {X 101.709,Y 85.509,Z 72.469,A 180.000,B 0.000,C 180.000} C_DIS
LIN {X 101.562,Y 85.460,Z 72.467,A 180.000,B 0.000,C 180.000} C_DIS
LIN {X 101.416,Y 85.412,Z 72.464,A 180.000,B 0.000,C 180.000} C_DIS
LIN {X 101.266,Y 85.363,Z 72.461,A 180.000,B 0.000,C 180.000} C_DIS
LIN {X 101.117,Y 85.314,Z 72.458,A 180.000,B 0.000,C 180.000} C_DIS
LIN {X 100.978,Y 85.271,Z 72.456,A 180.000,B 0.000,C 180.000} C_DIS
LIN {X 100.838,Y 85.233,Z 72.453,A 180.000,B 0.000,C 180.000} C_DIS
LIN {X 100.686,Y 85.192,Z 72.450,A 180.000,B 0.000,C 180.000} C_DIS
LIN {X 100.535,Y 85.151,Z 72.446,A 180.000,B 0.000,C 180.000} C_DIS
LIN {X 100.392,Y 85.113,Z 72.443,A 180.000,B 0.000,C 180.000} C_DIS
LIN {X 100.247,Y 85.080,Z 72.440,A 180.000,B 0.000,C 180.000} C_DIS
LIN {X 100.096,Y 85.048,Z 72.436,A 180.000,B 0.000,C 180.000} C_DIS
LIN {X 99.944,Y 85.016,Z 72.433,A 180.000,B 0.000,C 180.000} C_DIS
LIN {X 99.797,Y 84.985,Z 72.429,A 180.000,B 0.000,C 180.000} C_DIS
LIN {X 99.650,Y 84.955,Z 72.426,A 180.000,B 0.000,C 180.000} C_DIS
LIN {X 99.499,Y 84.930,Z 72.422,A 180.000,B 0.000,C 180.000} C_DIS
LIN {X 99.348,Y 84.906,Z 72.418,A 180.000,B 0.000,C 180.000} C_DIS
LIN {X 99.193,Y 84.883,Z 72.414,A 180.000,B 0.000,C 180.000} C_DIS
LIN {X 99.037,Y 84.859,Z 72.410,A 180.000,B 0.000,C 180.000} C_DIS
LIN {X 98.893,Y 84.839,Z 72.406,A 180.000,B 0.000,C 180.000} C_DIS
LIN {X 98.748,Y 84.825,Z 72.402,A 180.000,B 0.000,C 180.000} C_DIS
LIN {X 98.591,Y 84.810,Z 72.398,A 180.000,B 0.000,C 180.000} C_DIS
LIN {X 98.434,Y 84.794,Z 72.394,A 180.000,B 0.000,C 180.000} C_DIS
LIN {X 98.283,Y 84.780,Z 72.389,A 180.000,B 0.000,C 180.000} C_DIS
LIN {X 98.131,Y 84.769,Z 72.385,A 180.000,B 0.000,C 180.000} C_DIS
LIN {X 97.980,Y 84.763,Z 72.381,A 180.000,B 0.000,C 180.000} C_DIS
LIN {X 97.829,Y 84.756,Z 72.376,A 180.000,B 0.000,C 180.000} C_DIS
LIN {X 97.675,Y 84.750,Z 72.372,A 180.000,B 0.000,C 180.000} C_DIS
LIN {X 97.522,Y 84.744,Z 72.367,A 180.000,B 0.000,C 180.000} C_DIS
LIN {X 97.372,Y 84.744,Z 72.362,A 180.000,B 0.000,C 180.000} C_DIS
LIN {X 97.221,Y 84.746,Z 72.358,A 180.000,B 0.000,C 180.000} C_DIS
LIN {X 97.066,Y 84.748,Z 72.353,A 180.000,B 0.000,C 180.000} C_DIS
LIN {X 96.911,Y 84.750,Z 72.348,A 180.000,B 0.000,C 180.000} C_DIS
LIN {X 96.762,Y 84.755,Z 72.343,A 180.000,B 0.000,C 180.000} C_DIS
LIN {X 96.612,Y 84.764,Z 72.338,A 180.000,B 0.000,C 180.000} C_DIS
LIN {X 96.534,Y 84.770,Z 72.335,A 180.000,B 0.000,C 180.000} C_DIS
LIN {X 96.456,Y 84.775,Z 72.333,A 180.000,B 0.000,C 180.000} C_DIS
LIN {X 96.378,Y 84.780,Z 72.330,A 180.000,B 0.000,C 180.000} C_DIS
LIN {X 96.299,Y 84.786,Z 72.328,A 180.000,B 0.000,C 180.000} C_DIS
LIN {X 96.152,Y 84.796,Z 72.322,A 180.000,B 0.000,C 180.000} C_DIS
LIN {X 96.079,Y 84.801,Z 72.320,A 180.000,B 0.000,C 180.000} C_DIS
LIN {X 96.006,Y 84.809,Z 72.317,A 180.000,B 0.000,C 180.000} C_DIS
LIN {X 95.928,Y 84.819,Z 72.315,A 180.000,B 0.000,C 180.000} C_DIS
LIN {X 95.850,Y 84.828,Z 72.312,A 180.000,B 0.000,C 180.000} C_DIS
LIN {X 95.540,Y 84.867,Z 72.301,A 180.000,B 0.000,C 180.000} C_DIS
LIN {X 95.463,Y 84.877,Z 72.298,A 180.000,B 0.000,C 180.000} C_DIS
LIN {X 95.386,Y 84.887,Z 72.296,A 180.000,B 0.000,C 180.000} C_DIS
LIN {X 95.312,Y 84.899,Z 72.293,A 180.000,B 0.000,C 180.000} C_DIS
LIN {X 95.239,Y 84.912,Z 72.290,A 180.000,B 0.000,C 180.000} C_DIS
LIN {X 95.015,Y 84.953,Z 72.283,A 180.000,B 0.000,C 180.000} C_DIS
LIN {X 94.860,Y 84.981,Z 72.277,A 180.000,B 0.000,C 180.000} C_DIS
LIN {X 94.783,Y 84.995,Z 72.274,A 180.000,B 0.000,C 180.000} C_DIS
LIN {X 94.710,Y 85.008,Z 72.272,A 180.000,B 0.000,C 180.000} C_DIS
LIN {X 94.636,Y 85.023,Z 72.269,A 180.000,B 0.000,C 180.000} C_DIS
LIN {X 94.564,Y 85.039,Z 72.266,A 180.000,B 0.000,C 180.000} C_DIS
LIN {X 94.491,Y 85.057,Z 72.264,A 180.000,B 0.000,C 180.000} C_DIS
LIN {X 94.339,Y 85.093,Z 72.258,A 180.000,B 0.000,C 180.000} C_DIS
LIN {X 94.115,Y 85.147,Z 72.250,A 180.000,B 0.000,C 180.000} C_DIS
LIN {X 94.043,Y 85.165,Z 72.248,A 180.000,B 0.000,C 180.000} C_DIS
LIN {X 93.971,Y 85.183,Z 72.245,A 180.000,B 0.000,C 180.000} C_DIS
LIN {X 93.900,Y 85.203,Z 72.243,A 180.000,B 0.000,C 180.000} C_DIS
LIN {X 93.749,Y 85.248,Z 72.237,A 180.000,B 0.000,C 180.000} C_DIS
LIN {X 93.524,Y 85.316,Z 72.229,A 180.000,B 0.000,C 180.000} C_DIS
LIN {X 93.374,Y 85.361,Z 72.223,A 180.000,B 0.000,C 180.000} C_DIS
LIN {X 93.300,Y 85.384,Z 72.221,A 180.000,B 0.000,C 180.000} C_DIS
LIN {X 93.229,Y 85.407,Z 72.218,A 180.000,B 0.000,C 180.000} C_DIS
LIN {X 93.158,Y 85.432,Z 72.215,A 180.000,B 0.000,C 180.000} C_DIS
LIN {X 92.724,Y 85.590,Z 72.199,A 180.000,B 0.000,C 180.000} C_DIS
LIN {X 92.654,Y 85.615,Z 72.197,A 180.000,B 0.000,C 180.000} C_DIS
LIN {X 92.584,Y 85.642,Z 72.194,A 180.000,B 0.000,C 180.000} C_DIS
LIN {X 92.515,Y 85.671,Z 72.192,A 180.000,B 0.000,C 180.000} C_DIS
LIN {X 92.446,Y 85.700,Z 72.189,A 180.000,B 0.000,C 180.000} C_DIS
LIN {X 92.301,Y 85.762,Z 72.183,A 180.000,B 0.000,C 180.000} C_DIS
LIN {X 92.087,Y 85.854,Z 72.175,A 180.000,B 0.000,C 180.000} C_DIS
LIN {X 92.016,Y 85.884,Z 72.173,A 180.000,B 0.000,C 180.000} C_DIS
LIN {X 91.947,Y 85.915,Z 72.170,A 180.000,B 0.000,C 180.000} C_DIS
LIN {X 91.877,Y 85.947,Z 72.167,A 180.000,B 0.000,C 180.000} C_DIS
LIN {X 91.808,Y 85.981,Z 72.165,A 180.000,B 0.000,C 180.000} C_DIS
LIN {X 91.671,Y 86.049,Z 72.159,A 180.000,B 0.000,C 180.000} C_DIS
LIN {X 91.602,Y 86.083,Z 72.157,A 180.000,B 0.000,C 180.000} C_DIS
LIN {X 91.461,Y 86.153,Z 72.151,A 180.000,B 0.000,C 180.000} C_DIS
LIN {X 91.390,Y 86.188,Z 72.148,A 180.000,B 0.000,C 180.000} C_DIS
LIN {X 91.320,Y 86.223,Z 72.146,A 180.000,B 0.000,C 180.000} C_DIS
LIN {X 91.254,Y 86.258,Z 72.143,A 180.000,B 0.000,C 180.000} C_DIS
LIN {X 91.189,Y 86.295,Z 72.140,A 180.000,B 0.000,C 180.000} C_DIS
LIN {X 90.787,Y 86.523,Z 72.124,A 180.000,B 0.000,C 180.000} C_DIS
LIN {X 90.722,Y 86.560,Z 72.122,A 180.000,B 0.000,C 180.000} C_DIS
LIN {X 90.657,Y 86.599,Z 72.119,A 180.000,B 0.000,C 180.000} C_DIS
LIN {X 90.592,Y 86.639,Z 72.116,A 180.000,B 0.000,C 180.000} C_DIS
LIN {X 90.529,Y 86.679,Z 72.114,A 180.000,B 0.000,C 180.000} C_DIS
LIN {X 90.331,Y 86.807,Z 72.105,A 180.000,B 0.000,C 180.000} C_DIS
LIN {X 90.137,Y 86.932,Z 72.097,A 180.000,B 0.000,C 180.000} C_DIS
LIN {X 90.074,Y 86.973,Z 72.095,A 180.000,B 0.000,C 180.000} C_DIS
LIN {X 90.011,Y 87.016,Z 72.092,A 180.000,B 0.000,C 180.000} C_DIS
LIN {X 89.948,Y 87.062,Z 72.089,A 180.000,B 0.000,C 180.000} C_DIS
LIN {X 89.572,Y 87.335,Z 72.073,A 180.000,B 0.000,C 180.000} C_DIS
LIN {X 89.509,Y 87.381,Z 72.070,A 180.000,B 0.000,C 180.000} C_DIS
LIN {X 89.449,Y 87.427,Z 72.068,A 180.000,B 0.000,C 180.000} C_DIS
LIN {X 89.389,Y 87.475,Z 72.065,A 180.000,B 0.000,C 180.000} C_DIS
LIN {X 89.330,Y 87.524,Z 72.062,A 180.000,B 0.000,C 180.000} C_DIS
LIN {X 89.026,Y 87.771,Z 72.049,A 180.000,B 0.000,C 180.000} C_DIS
LIN {X 88.968,Y 87.819,Z 72.046,A 180.000,B 0.000,C 180.000} C_DIS
LIN {X 88.910,Y 87.867,Z 72.043,A 180.000,B 0.000,C 180.000} C_DIS
LIN {X 88.853,Y 87.916,Z 72.041,A 180.000,B 0.000,C 180.000} C_DIS
